KUKA KRL program: sKontur5.src, sKontur5.dat

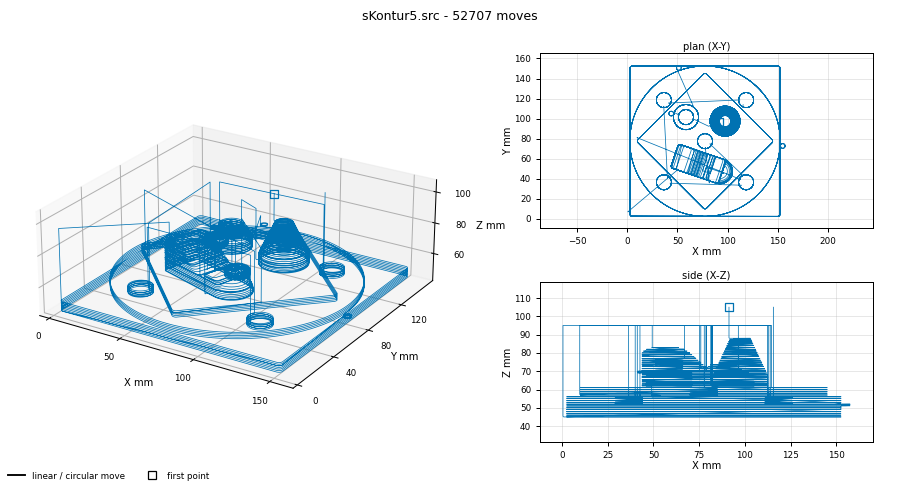
[picture p0: tool path of sKontur5.src, 52707 of 52708 moves have a stored position in this frame; points joined in program order, loops and branches not executed]
--- sKontur5.src ---
&ACCESS RVO
DEF sKontur5()
; Generated by AUTODESK Fusion 360 CAM 2.0.14793
; Creation date: Thursday, March 16, 2023 18:51:27
;FOLD sKontur5
; Start position (joint) = {A1 5,A2 -80,A3 100,A4 75,A5 -60,A6 -65}
; Tool Number            = 4
; Base Number            = 1
; Spindle Speed          = 5000 RPM
; Program file name      = sKontur5.src

PTP {A1 5,A2 -80,A3 100,A4 75,A5 -60,A6 -65,E1 0,E2 0,E3 0,E4 0,E5 0,E6 0}
LIN {X 91.288,Y 96.306,Z 105.000,A 180.000,B 0.000,C 180.000} C_DIS
LIN {X 91.288,Y 96.306,Z 90.497,A 180.000,B 0.000,C 180.000} C_DIS
; Plunge Move Starts
$VEL.CP=0.01
LIN {X 91.288,Y 96.306,Z 89.476,A 180.000,B 0.000,C 180.000} C_DIS
; Lead In Move Starts
LIN {X 91.288,Y 96.306,Z 88.351,A 180.000,B 0.000,C 180.000} C_DIS
LIN {X 91.390,Y 96.319,Z 88.103,A 180.000,B 0.000,C 180.000} C_DIS
LIN {X 91.636,Y 96.350,Z 88.000,A 180.000,B 0.000,C 180.000} C_DIS
LIN {X 91.969,Y 96.540,Z 88.000,A 180.000,B 0.000,C 180.000} C_DIS
LIN {X 92.070,Y 96.909,Z 88.000,A 180.000,B 0.000,C 180.000} C_DIS
; Cutting Move Starts
$VEL.CP=0.02
LIN {X 92.051,Y 97.075,Z 88.000,A 180.000,B 0.000,C 180.000} C_DIS
LIN {X 92.040,Y 97.254,Z 88.000,A 180.000,B 0.000,C 180.000} C_DIS
LIN {X 92.038,Y 97.433,Z 88.000,A 180.000,B 0.000,C 180.000} C_DIS
LIN {X 92.038,Y 97.612,Z 88.000,A 180.000,B 0.000,C 180.000} C_DIS
LIN {X 92.042,Y 97.790,Z 88.000,A 180.000,B 0.000,C 180.000} C_DIS
LIN {X 92.055,Y 97.969,Z 88.000,A 180.000,B 0.000,C 180.000} C_DIS
LIN {X 92.070,Y 98.091,Z 88.000,A 180.000,B 0.000,C 180.000} C_DIS
LIN {X 92.099,Y 98.327,Z 88.000,A 180.000,B 0.000,C 180.000} C_DIS
LIN {X 92.127,Y 98.505,Z 88.000,A 180.000,B 0.000,C 180.000} C_DIS
LIN {X 92.166,Y 98.684,Z 88.000,A 180.000,B 0.000,C 180.000} C_DIS
LIN {X 92.211,Y 98.863,Z 88.000,A 180.000,B 0.000,C 180.000} C_DIS
LIN {X 92.249,Y 99.007,Z 88.000,A 180.000,B 0.000,C 180.000} C_DIS
LIN {X 92.257,Y 99.042,Z 88.000,A 180.000,B 0.000,C 180.000} C_DIS
LIN {X 92.312,Y 99.221,Z 88.000,A 180.000,B 0.000,C 180.000} C_DIS
LIN {X 92.378,Y 99.399,Z 88.000,A 180.000,B 0.000,C 180.000} C_DIS
LIN {X 92.449,Y 99.578,Z 88.000,A 180.000,B 0.000,C 180.000} C_DIS
LIN {X 92.522,Y 99.757,Z 88.000,A 180.000,B 0.000,C 180.000} C_DIS
LIN {X 92.606,Y 99.932,Z 88.000,A 180.000,B 0.000,C 180.000} C_DIS
LIN {X 92.608,Y 99.936,Z 88.000,A 180.000,B 0.000,C 180.000} C_DIS
LIN {X 92.705,Y 100.114,Z 88.000,A 180.000,B 0.000,C 180.000} C_DIS
LIN {X 92.785,Y 100.260,Z 88.000,A 180.000,B 0.000,C 180.000} C_DIS
LIN {X 92.803,Y 100.293,Z 88.000,A 180.000,B 0.000,C 180.000} C_DIS
LIN {X 92.913,Y 100.472,Z 88.000,A 180.000,B 0.000,C 180.000} C_DIS
LIN {X 92.964,Y 100.547,Z 88.000,A 180.000,B 0.000,C 180.000} C_DIS
LIN {X 93.038,Y 100.651,Z 88.000,A 180.000,B 0.000,C 180.000} C_DIS
LIN {X 93.168,Y 100.829,Z 88.000,A 180.000,B 0.000,C 180.000} C_DIS
LIN {X 93.308,Y 101.008,Z 88.000,A 180.000,B 0.000,C 180.000} C_DIS
LIN {X 93.321,Y 101.023,Z 88.000,A 180.000,B 0.000,C 180.000} C_DIS
LIN {X 93.470,Y 101.187,Z 88.000,A 180.000,B 0.000,C 180.000} C_DIS
LIN {X 93.500,Y 101.218,Z 88.000,A 180.000,B 0.000,C 180.000} C_DIS
LIN {X 93.638,Y 101.366,Z 88.000,A 180.000,B 0.000,C 180.000} C_DIS
LIN {X 93.679,Y 101.407,Z 88.000,A 180.000,B 0.000,C 180.000} C_DIS
LIN {X 93.824,Y 101.545,Z 88.000,A 180.000,B 0.000,C 180.000} C_DIS
LIN {X 93.857,Y 101.574,Z 88.000,A 180.000,B 0.000,C 180.000} C_DIS
LIN {X 94.037,Y 101.723,Z 88.000,A 180.000,B 0.000,C 180.000} C_DIS
LIN {X 94.215,Y 101.868,Z 88.000,A 180.000,B 0.000,C 180.000} C_DIS
LIN {X 94.260,Y 101.902,Z 88.000,A 180.000,B 0.000,C 180.000} C_DIS
LIN {X 94.394,Y 101.996,Z 88.000,A 180.000,B 0.000,C 180.000} C_DIS
LIN {X 94.525,Y 102.081,Z 88.000,A 180.000,B 0.000,C 180.000} C_DIS
LIN {X 94.573,Y 102.111,Z 88.000,A 180.000,B 0.000,C 180.000} C_DIS
LIN {X 94.751,Y 102.223,Z 88.000,A 180.000,B 0.000,C 180.000} C_DIS
LIN {X 94.813,Y 102.260,Z 88.000,A 180.000,B 0.000,C 180.000} C_DIS
LIN {X 94.930,Y 102.324,Z 88.000,A 180.000,B 0.000,C 180.000} C_DIS
LIN {X 95.109,Y 102.411,Z 88.000,A 180.000,B 0.000,C 180.000} C_DIS
LIN {X 95.288,Y 102.495,Z 88.000,A 180.000,B 0.000,C 180.000} C_DIS
LIN {X 95.466,Y 102.574,Z 88.000,A 180.000,B 0.000,C 180.000} C_DIS
LIN {X 95.580,Y 102.617,Z 88.000,A 180.000,B 0.000,C 180.000} C_DIS
LIN {X 95.645,Y 102.640,Z 88.000,A 180.000,B 0.000,C 180.000} C_DIS
LIN {X 95.824,Y 102.698,Z 88.000,A 180.000,B 0.000,C 180.000} C_DIS
LIN {X 96.003,Y 102.756,Z 88.000,A 180.000,B 0.000,C 180.000} C_DIS
LIN {X 96.147,Y 102.796,Z 88.000,A 180.000,B 0.000,C 180.000} C_DIS
LIN {X 96.181,Y 102.805,Z 88.000,A 180.000,B 0.000,C 180.000} C_DIS
LIN {X 96.360,Y 102.843,Z 88.000,A 180.000,B 0.000,C 180.000} C_DIS
LIN {X 96.539,Y 102.877,Z 88.000,A 180.000,B 0.000,C 180.000} C_DIS
LIN {X 96.718,Y 102.909,Z 88.000,A 180.000,B 0.000,C 180.000} C_DIS
LIN {X 96.897,Y 102.932,Z 88.000,A 180.000,B 0.000,C 180.000} C_DIS
LIN {X 97.075,Y 102.946,Z 88.000,A 180.000,B 0.000,C 180.000} C_DIS
LIN {X 97.254,Y 102.957,Z 88.000,A 180.000,B 0.000,C 180.000} C_DIS
LIN {X 97.433,Y 102.965,Z 88.000,A 180.000,B 0.000,C 180.000} C_DIS
LIN {X 97.612,Y 102.964,Z 88.000,A 180.000,B 0.000,C 180.000} C_DIS
LIN {X 97.790,Y 102.954,Z 88.000,A 180.000,B 0.000,C 180.000} C_DIS
LIN {X 97.969,Y 102.943,Z 88.000,A 180.000,B 0.000,C 180.000} C_DIS
LIN {X 98.148,Y 102.928,Z 88.000,A 180.000,B 0.000,C 180.000} C_DIS
LIN {X 98.327,Y 102.902,Z 88.000,A 180.000,B 0.000,C 180.000} C_DIS
LIN {X 98.505,Y 102.868,Z 88.000,A 180.000,B 0.000,C 180.000} C_DIS
LIN {X 98.684,Y 102.834,Z 88.000,A 180.000,B 0.000,C 180.000} C_DIS
LIN {X 98.853,Y 102.796,Z 88.000,A 180.000,B 0.000,C 180.000} C_DIS
LIN {X 98.863,Y 102.793,Z 88.000,A 180.000,B 0.000,C 180.000} C_DIS
LIN {X 99.042,Y 102.742,Z 88.000,A 180.000,B 0.000,C 180.000} C_DIS
LIN {X 99.221,Y 102.683,Z 88.000,A 180.000,B 0.000,C 180.000} C_DIS
LIN {X 99.399,Y 102.625,Z 88.000,A 180.000,B 0.000,C 180.000} C_DIS
LIN {X 99.420,Y 102.617,Z 88.000,A 180.000,B 0.000,C 180.000} C_DIS
LIN {X 99.578,Y 102.555,Z 88.000,A 180.000,B 0.000,C 180.000} C_DIS
LIN {X 99.757,Y 102.474,Z 88.000,A 180.000,B 0.000,C 180.000} C_DIS
LIN {X 99.936,Y 102.390,Z 88.000,A 180.000,B 0.000,C 180.000} C_DIS
LIN {X 100.114,Y 102.300,Z 88.000,A 180.000,B 0.000,C 180.000} C_DIS
LIN {X 100.187,Y 102.260,Z 88.000,A 180.000,B 0.000,C 180.000} C_DIS
LIN {X 100.293,Y 102.196,Z 88.000,A 180.000,B 0.000,C 180.000} C_DIS
LIN {X 100.475,Y 102.081,Z 88.000,A 180.000,B 0.000,C 180.000} C_DIS
LIN {X 100.651,Y 101.966,Z 88.000,A 180.000,B 0.000,C 180.000} C_DIS
LIN {X 100.740,Y 101.902,Z 88.000,A 180.000,B 0.000,C 180.000} C_DIS
LIN {X 100.829,Y 101.833,Z 88.000,A 180.000,B 0.000,C 180.000} C_DIS
LIN {X 100.963,Y 101.723,Z 88.000,A 180.000,B 0.000,C 180.000} C_DIS
LIN {X 101.008,Y 101.686,Z 88.000,A 180.000,B 0.000,C 180.000} C_DIS
LIN {X 101.176,Y 101.545,Z 88.000,A 180.000,B 0.000,C 180.000} C_DIS
LIN {X 101.187,Y 101.535,Z 88.000,A 180.000,B 0.000,C 180.000} C_DIS
LIN {X 101.362,Y 101.366,Z 88.000,A 180.000,B 0.000,C 180.000} C_DIS
LIN {X 101.366,Y 101.361,Z 88.000,A 180.000,B 0.000,C 180.000} C_DIS
LIN {X 101.530,Y 101.187,Z 88.000,A 180.000,B 0.000,C 180.000} C_DIS
LIN {X 101.545,Y 101.171,Z 88.000,A 180.000,B 0.000,C 180.000} C_DIS
LIN {X 101.692,Y 101.008,Z 88.000,A 180.000,B 0.000,C 180.000} C_DIS
LIN {X 101.723,Y 100.970,Z 88.000,A 180.000,B 0.000,C 180.000} C_DIS
LIN {X 101.832,Y 100.829,Z 88.000,A 180.000,B 0.000,C 180.000} C_DIS
LIN {X 101.962,Y 100.651,Z 88.000,A 180.000,B 0.000,C 180.000} C_DIS
LIN {X 102.081,Y 100.482,Z 88.000,A 180.000,B 0.000,C 180.000} C_DIS
LIN {X 102.087,Y 100.472,Z 88.000,A 180.000,B 0.000,C 180.000} C_DIS
LIN {X 102.197,Y 100.293,Z 88.000,A 180.000,B 0.000,C 180.000} C_DIS
LIN {X 102.260,Y 100.179,Z 88.000,A 180.000,B 0.000,C 180.000} C_DIS
LIN {X 102.295,Y 100.114,Z 88.000,A 180.000,B 0.000,C 180.000} C_DIS
LIN {X 102.392,Y 99.936,Z 88.000,A 180.000,B 0.000,C 180.000} C_DIS
LIN {X 102.438,Y 99.844,Z 88.000,A 180.000,B 0.000,C 180.000} C_DIS
LIN {X 102.478,Y 99.757,Z 88.000,A 180.000,B 0.000,C 180.000} C_DIS
LIN {X 102.551,Y 99.578,Z 88.000,A 180.000,B 0.000,C 180.000} C_DIS
LIN {X 102.622,Y 99.399,Z 88.000,A 180.000,B 0.000,C 180.000} C_DIS
LIN {X 102.688,Y 99.221,Z 88.000,A 180.000,B 0.000,C 180.000} C_DIS
LIN {X 102.743,Y 99.042,Z 88.000,A 180.000,B 0.000,C 180.000} C_DIS
LIN {X 102.789,Y 98.863,Z 88.000,A 180.000,B 0.000,C 180.000} C_DIS
LIN {X 102.796,Y 98.834,Z 88.000,A 180.000,B 0.000,C 180.000} C_DIS
LIN {X 102.834,Y 98.684,Z 88.000,A 180.000,B 0.000,C 180.000} C_DIS
LIN {X 102.873,Y 98.505,Z 88.000,A 180.000,B 0.000,C 180.000} C_DIS
LIN {X 102.901,Y 98.327,Z 88.000,A 180.000,B 0.000,C 180.000} C_DIS
LIN {X 102.923,Y 98.148,Z 88.000,A 180.000,B 0.000,C 180.000} C_DIS
LIN {X 102.945,Y 97.969,Z 88.000,A 180.000,B 0.000,C 180.000} C_DIS
LIN {X 102.958,Y 97.790,Z 88.000,A 180.000,B 0.000,C 180.000} C_DIS
LIN {X 102.962,Y 97.612,Z 88.000,A 180.000,B 0.000,C 180.000} C_DIS
LIN {X 102.962,Y 97.433,Z 88.000,A 180.000,B 0.000,C 180.000} C_DIS
LIN {X 102.960,Y 97.254,Z 88.000,A 180.000,B 0.000,C 180.000} C_DIS
LIN {X 102.949,Y 97.075,Z 88.000,A 180.000,B 0.000,C 180.000} C_DIS
LIN {X 102.929,Y 96.897,Z 88.000,A 180.000,B 0.000,C 180.000} C_DIS
LIN {X 102.906,Y 96.718,Z 88.000,A 180.000,B 0.000,C 180.000} C_DIS
LIN {X 102.881,Y 96.539,Z 88.000,A 180.000,B 0.000,C 180.000} C_DIS
LIN {X 102.845,Y 96.360,Z 88.000,A 180.000,B 0.000,C 180.000} C_DIS
LIN {X 102.800,Y 96.181,Z 88.000,A 180.000,B 0.000,C 180.000} C_DIS
LIN {X 102.754,Y 96.003,Z 88.000,A 180.000,B 0.000,C 180.000} C_DIS
LIN {X 102.703,Y 95.824,Z 88.000,A 180.000,B 0.000,C 180.000} C_DIS
LIN {X 102.639,Y 95.645,Z 88.000,A 180.000,B 0.000,C 180.000} C_DIS
LIN {X 102.617,Y 95.588,Z 88.000,A 180.000,B 0.000,C 180.000} C_DIS
LIN {X 102.569,Y 95.466,Z 88.000,A 180.000,B 0.000,C 180.000} C_DIS
LIN {X 102.497,Y 95.288,Z 88.000,A 180.000,B 0.000,C 180.000} C_DIS
LIN {X 102.438,Y 95.156,Z 88.000,A 180.000,B 0.000,C 180.000} C_DIS
LIN {X 102.415,Y 95.109,Z 88.000,A 180.000,B 0.000,C 180.000} C_DIS
LIN {X 102.320,Y 94.930,Z 88.000,A 180.000,B 0.000,C 180.000} C_DIS
LIN {X 102.221,Y 94.751,Z 88.000,A 180.000,B 0.000,C 180.000} C_DIS
LIN {X 102.116,Y 94.573,Z 88.000,A 180.000,B 0.000,C 180.000} C_DIS
LIN {X 102.081,Y 94.518,Z 88.000,A 180.000,B 0.000,C 180.000} C_DIS
LIN {X 101.994,Y 94.394,Z 88.000,A 180.000,B 0.000,C 180.000} C_DIS
LIN {X 101.864,Y 94.215,Z 88.000,A 180.000,B 0.000,C 180.000} C_DIS
LIN {X 101.729,Y 94.036,Z 88.000,A 180.000,B 0.000,C 180.000} C_DIS
LIN {X 101.723,Y 94.030,Z 88.000,A 180.000,B 0.000,C 180.000} C_DIS
LIN {X 101.571,Y 93.857,Z 88.000,A 180.000,B 0.000,C 180.000} C_DIS
LIN {X 101.404,Y 93.679,Z 88.000,A 180.000,B 0.000,C 180.000} C_DIS
LIN {X 101.366,Y 93.639,Z 88.000,A 180.000,B 0.000,C 180.000} C_DIS
LIN {X 101.225,Y 93.500,Z 88.000,A 180.000,B 0.000,C 180.000} C_DIS
LIN {X 101.187,Y 93.465,Z 88.000,A 180.000,B 0.000,C 180.000} C_DIS
LIN {X 101.017,Y 93.321,Z 88.000,A 180.000,B 0.000,C 180.000} C_DIS
LIN {X 101.008,Y 93.314,Z 88.000,A 180.000,B 0.000,C 180.000} C_DIS
LIN {X 100.829,Y 93.167,Z 88.000,A 180.000,B 0.000,C 180.000} C_DIS
LIN {X 100.799,Y 93.142,Z 88.000,A 180.000,B 0.000,C 180.000} C_DIS
LIN {X 100.651,Y 93.034,Z 88.000,A 180.000,B 0.000,C 180.000} C_DIS
LIN {X 100.545,Y 92.964,Z 88.000,A 180.000,B 0.000,C 180.000} C_DIS
LIN {X 100.293,Y 92.804,Z 88.000,A 180.000,B 0.000,C 180.000} C_DIS
LIN {X 100.262,Y 92.785,Z 88.000,A 180.000,B 0.000,C 180.000} C_DIS
LIN {X 100.114,Y 92.700,Z 88.000,A 180.000,B 0.000,C 180.000} C_DIS
LIN {X 99.936,Y 92.610,Z 88.000,A 180.000,B 0.000,C 180.000} C_DIS
LIN {X 99.757,Y 92.526,Z 88.000,A 180.000,B 0.000,C 180.000} C_DIS
LIN {X 99.578,Y 92.445,Z 88.000,A 180.000,B 0.000,C 180.000} C_DIS
LIN {X 99.537,Y 92.427,Z 88.000,A 180.000,B 0.000,C 180.000} C_DIS
LIN {X 99.399,Y 92.375,Z 88.000,A 180.000,B 0.000,C 180.000} C_DIS
LIN {X 99.221,Y 92.317,Z 88.000,A 180.000,B 0.000,C 180.000} C_DIS
LIN {X 99.042,Y 92.258,Z 88.000,A 180.000,B 0.000,C 180.000} C_DIS
LIN {X 99.010,Y 92.249,Z 88.000,A 180.000,B 0.000,C 180.000} C_DIS
LIN {X 98.863,Y 92.207,Z 88.000,A 180.000,B 0.000,C 180.000} C_DIS
LIN {X 98.684,Y 92.166,Z 88.000,A 180.000,B 0.000,C 180.000} C_DIS
LIN {X 98.505,Y 92.132,Z 88.000,A 180.000,B 0.000,C 180.000} C_DIS
LIN {X 98.327,Y 92.098,Z 88.000,A 180.000,B 0.000,C 180.000} C_DIS
LIN {X 98.148,Y 92.072,Z 88.000,A 180.000,B 0.000,C 180.000} C_DIS
LIN {X 98.124,Y 92.070,Z 88.000,A 180.000,B 0.000,C 180.000} C_DIS
LIN {X 97.969,Y 92.057,Z 88.000,A 180.000,B 0.000,C 180.000} C_DIS
LIN {X 97.790,Y 92.046,Z 88.000,A 180.000,B 0.000,C 180.000} C_DIS
LIN {X 97.612,Y 92.036,Z 88.000,A 180.000,B 0.000,C 180.000} C_DIS
LIN {X 97.433,Y 92.035,Z 88.000,A 180.000,B 0.000,C 180.000} C_DIS
LIN {X 97.254,Y 92.043,Z 88.000,A 180.000,B 0.000,C 180.000} C_DIS
LIN {X 97.075,Y 92.054,Z 88.000,A 180.000,B 0.000,C 180.000} C_DIS
LIN {X 96.897,Y 92.068,Z 88.000,A 180.000,B 0.000,C 180.000} C_DIS
LIN {X 96.876,Y 92.070,Z 88.000,A 180.000,B 0.000,C 180.000} C_DIS
LIN {X 96.718,Y 92.091,Z 88.000,A 180.000,B 0.000,C 180.000} C_DIS
LIN {X 96.539,Y 92.123,Z 88.000,A 180.000,B 0.000,C 180.000} C_DIS
LIN {X 96.360,Y 92.157,Z 88.000,A 180.000,B 0.000,C 180.000} C_DIS
LIN {X 96.181,Y 92.195,Z 88.000,A 180.000,B 0.000,C 180.000} C_DIS
LIN {X 96.003,Y 92.244,Z 88.000,A 180.000,B 0.000,C 180.000} C_DIS
LIN {X 95.990,Y 92.249,Z 88.000,A 180.000,B 0.000,C 180.000} C_DIS
LIN {X 95.824,Y 92.302,Z 88.000,A 180.000,B 0.000,C 180.000} C_DIS
LIN {X 95.645,Y 92.360,Z 88.000,A 180.000,B 0.000,C 180.000} C_DIS
LIN {X 95.466,Y 92.426,Z 88.000,A 180.000,B 0.000,C 180.000} C_DIS
LIN {X 95.463,Y 92.427,Z 88.000,A 180.000,B 0.000,C 180.000} C_DIS
LIN {X 95.288,Y 92.505,Z 88.000,A 180.000,B 0.000,C 180.000} C_DIS
LIN {X 95.073,Y 92.606,Z 88.000,A 180.000,B 0.000,C 180.000} C_DIS
LIN {X 94.930,Y 92.676,Z 88.000,A 180.000,B 0.000,C 180.000} C_DIS
LIN {X 94.751,Y 92.777,Z 88.000,A 180.000,B 0.000,C 180.000} C_DIS
LIN {X 94.738,Y 92.785,Z 88.000,A 180.000,B 0.000,C 180.000} C_DIS
LIN {X 94.573,Y 92.889,Z 88.000,A 180.000,B 0.000,C 180.000} C_DIS
LIN {X 94.455,Y 92.964,Z 88.000,A 180.000,B 0.000,C 180.000} C_DIS
LIN {X 94.394,Y 93.004,Z 88.000,A 180.000,B 0.000,C 180.000} C_DIS
LIN {X 94.215,Y 93.132,Z 88.000,A 180.000,B 0.000,C 180.000} C_DIS
LIN {X 94.201,Y 93.142,Z 88.000,A 180.000,B 0.000,C 180.000} C_DIS
LIN {X 94.036,Y 93.277,Z 88.000,A 180.000,B 0.000,C 180.000} C_DIS
LIN {X 93.983,Y 93.321,Z 88.000,A 180.000,B 0.000,C 180.000} C_DIS
LIN {X 93.857,Y 93.426,Z 88.000,A 180.000,B 0.000,C 180.000} C_DIS
LIN {X 93.775,Y 93.500,Z 88.000,A 180.000,B 0.000,C 180.000} C_DIS
LIN {X 93.679,Y 93.593,Z 88.000,A 180.000,B 0.000,C 180.000} C_DIS
LIN {X 93.596,Y 93.679,Z 88.000,A 180.000,B 0.000,C 180.000} C_DIS
LIN {X 93.429,Y 93.857,Z 88.000,A 180.000,B 0.000,C 180.000} C_DIS
LIN {X 93.321,Y 93.977,Z 88.000,A 180.000,B 0.000,C 180.000} C_DIS
LIN {X 93.271,Y 94.036,Z 88.000,A 180.000,B 0.000,C 180.000} C_DIS
LIN {X 93.142,Y 94.206,Z 88.000,A 180.000,B 0.000,C 180.000} C_DIS
LIN {X 93.006,Y 94.394,Z 88.000,A 180.000,B 0.000,C 180.000} C_DIS
LIN {X 92.964,Y 94.453,Z 88.000,A 180.000,B 0.000,C 180.000} C_DIS
LIN {X 92.884,Y 94.573,Z 88.000,A 180.000,B 0.000,C 180.000} C_DIS
LIN {X 92.785,Y 94.740,Z 88.000,A 180.000,B 0.000,C 180.000} C_DIS
LIN {X 92.680,Y 94.930,Z 88.000,A 180.000,B 0.000,C 180.000} C_DIS
LIN {X 92.606,Y 95.068,Z 88.000,A 180.000,B 0.000,C 180.000} C_DIS
LIN {X 92.585,Y 95.109,Z 88.000,A 180.000,B 0.000,C 180.000} C_DIS
LIN {X 92.503,Y 95.288,Z 88.000,A 180.000,B 0.000,C 180.000} C_DIS
LIN {X 92.431,Y 95.466,Z 88.000,A 180.000,B 0.000,C 180.000} C_DIS
LIN {X 92.427,Y 95.476,Z 88.000,A 180.000,B 0.000,C 180.000} C_DIS
LIN {X 92.361,Y 95.645,Z 88.000,A 180.000,B 0.000,C 180.000} C_DIS
LIN {X 92.297,Y 95.824,Z 88.000,A 180.000,B 0.000,C 180.000} C_DIS
LIN {X 92.249,Y 95.993,Z 88.000,A 180.000,B 0.000,C 180.000} C_DIS
LIN {X 92.246,Y 96.003,Z 88.000,A 180.000,B 0.000,C 180.000} C_DIS
LIN {X 92.200,Y 96.181,Z 88.000,A 180.000,B 0.000,C 180.000} C_DIS
LIN {X 92.155,Y 96.360,Z 88.000,A 180.000,B 0.000,C 180.000} C_DIS
LIN {X 92.119,Y 96.539,Z 88.000,A 180.000,B 0.000,C 180.000} C_DIS
LIN {X 92.094,Y 96.718,Z 88.000,A 180.000,B 0.000,C 180.000} C_DIS
LIN {X 92.070,Y 96.909,Z 88.000,A 180.000,B 0.000,C 180.000} C_DIS
; Link Move Starts
LIN {X 92.043,Y 97.188,Z 88.000,A 180.000,B 0.000,C 180.000} C_DIS
LIN {X 92.038,Y 97.479,Z 87.999,A 180.000,B 0.000,C 180.000} C_DIS
LIN {X 92.040,Y 97.771,Z 87.998,A 180.000,B 0.000,C 180.000} C_DIS
LIN {X 92.064,Y 98.056,Z 87.997,A 180.000,B 0.000,C 180.000} C_DIS
LIN {X 92.101,Y 98.357,Z 87.995,A 180.000,B 0.000,C 180.000} C_DIS
LIN {X 92.148,Y 98.627,Z 87.993,A 180.000,B 0.000,C 180.000} C_DIS
LIN {X 92.221,Y 98.920,Z 87.990,A 180.000,B 0.000,C 180.000} C_DIS
LIN {X 92.298,Y 99.199,Z 87.987,A 180.000,B 0.000,C 180.000} C_DIS
LIN {X 92.396,Y 99.465,Z 87.984,A 180.000,B 0.000,C 180.000} C_DIS
LIN {X 92.506,Y 99.743,Z 87.980,A 180.000,B 0.000,C 180.000} C_DIS
LIN {X 92.627,Y 99.996,Z 87.976,A 180.000,B 0.000,C 180.000} C_DIS
LIN {X 92.770,Y 100.260,Z 87.972,A 180.000,B 0.000,C 180.000} C_DIS
LIN {X 92.916,Y 100.505,Z 87.967,A 180.000,B 0.000,C 180.000} C_DIS
LIN {X 93.000,Y 100.626,Z 87.964,A 180.000,B 0.000,C 180.000} C_DIS
LIN {X 93.086,Y 100.747,Z 87.962,A 180.000,B 0.000,C 180.000} C_DIS
LIN {X 93.171,Y 100.865,Z 87.959,A 180.000,B 0.000,C 180.000} C_DIS
LIN {X 93.259,Y 100.980,Z 87.956,A 180.000,B 0.000,C 180.000} C_DIS
LIN {X 93.351,Y 101.090,Z 87.954,A 180.000,B 0.000,C 180.000} C_DIS
LIN {X 93.448,Y 101.196,Z 87.951,A 180.000,B 0.000,C 180.000} C_DIS
LIN {X 93.547,Y 101.304,Z 87.948,A 180.000,B 0.000,C 180.000} C_DIS
LIN {X 93.646,Y 101.411,Z 87.945,A 180.000,B 0.000,C 180.000} C_DIS
LIN {X 93.746,Y 101.511,Z 87.941,A 180.000,B 0.000,C 180.000} C_DIS
LIN {X 93.851,Y 101.606,Z 87.938,A 180.000,B 0.000,C 180.000} C_DIS
LIN {X 93.969,Y 101.707,Z 87.935,A 180.000,B 0.000,C 180.000} C_DIS
LIN {X 94.088,Y 101.807,Z 87.931,A 180.000,B 0.000,C 180.000} C_DIS
LIN {X 94.193,Y 101.894,Z 87.928,A 180.000,B 0.000,C 180.000} C_DIS
LIN {X 94.301,Y 101.976,Z 87.925,A 180.000,B 0.000,C 180.000} C_DIS
LIN {X 94.427,Y 102.062,Z 87.921,A 180.000,B 0.000,C 180.000} C_DIS
LIN {X 94.554,Y 102.145,Z 87.917,A 180.000,B 0.000,C 180.000} C_DIS
LIN {X 94.674,Y 102.223,Z 87.913,A 180.000,B 0.000,C 180.000} C_DIS
LIN {X 94.795,Y 102.298,Z 87.910,A 180.000,B 0.000,C 180.000} C_DIS
LIN {X 94.922,Y 102.369,Z 87.906,A 180.000,B 0.000,C 180.000} C_DIS
LIN {X 95.052,Y 102.435,Z 87.902,A 180.000,B 0.000,C 180.000} C_DIS
LIN {X 95.190,Y 102.502,Z 87.898,A 180.000,B 0.000,C 180.000} C_DIS
LIN {X 95.329,Y 102.569,Z 87.893,A 180.000,B 0.000,C 180.000} C_DIS
LIN {X 95.461,Y 102.627,Z 87.889,A 180.000,B 0.000,C 180.000} C_DIS
LIN {X 95.596,Y 102.680,Z 87.885,A 180.000,B 0.000,C 180.000} C_DIS
LIN {X 95.736,Y 102.728,Z 87.881,A 180.000,B 0.000,C 180.000} C_DIS
LIN {X 95.875,Y 102.775,Z 87.876,A 180.000,B 0.000,C 180.000} C_DIS
LIN {X 96.010,Y 102.820,Z 87.872,A 180.000,B 0.000,C 180.000} C_DIS
LIN {X 96.146,Y 102.859,Z 87.868,A 180.000,B 0.000,C 180.000} C_DIS
LIN {X 96.290,Y 102.894,Z 87.863,A 180.000,B 0.000,C 180.000} C_DIS
LIN {X 96.436,Y 102.924,Z 87.859,A 180.000,B 0.000,C 180.000} C_DIS
LIN {X 96.584,Y 102.955,Z 87.854,A 180.000,B 0.000,C 180.000} C_DIS
LIN {X 96.733,Y 102.983,Z 87.849,A 180.000,B 0.000,C 180.000} C_DIS
LIN {X 96.872,Y 103.003,Z 87.844,A 180.000,B 0.000,C 180.000} C_DIS
LIN {X 97.011,Y 103.017,Z 87.840,A 180.000,B 0.000,C 180.000} C_DIS
LIN {X 97.087,Y 103.022,Z 87.837,A 180.000,B 0.000,C 180.000} C_DIS
LIN {X 97.163,Y 103.028,Z 87.835,A 180.000,B 0.000,C 180.000} C_DIS
LIN {X 97.238,Y 103.034,Z 87.832,A 180.000,B 0.000,C 180.000} C_DIS
LIN {X 97.314,Y 103.040,Z 87.830,A 180.000,B 0.000,C 180.000} C_DIS
LIN {X 97.457,Y 103.048,Z 87.825,A 180.000,B 0.000,C 180.000} C_DIS
LIN {X 97.601,Y 103.048,Z 87.820,A 180.000,B 0.000,C 180.000} C_DIS
LIN {X 97.677,Y 103.047,Z 87.817,A 180.000,B 0.000,C 180.000} C_DIS
LIN {X 97.752,Y 103.043,Z 87.815,A 180.000,B 0.000,C 180.000} C_DIS
LIN {X 97.976,Y 103.033,Z 87.807,A 180.000,B 0.000,C 180.000} C_DIS
LIN {X 98.049,Y 103.029,Z 87.804,A 180.000,B 0.000,C 180.000} C_DIS
LIN {X 98.122,Y 103.023,Z 87.802,A 180.000,B 0.000,C 180.000} C_DIS
LIN {X 98.195,Y 103.016,Z 87.799,A 180.000,B 0.000,C 180.000} C_DIS
LIN {X 98.267,Y 103.007,Z 87.797,A 180.000,B 0.000,C 180.000} C_DIS
LIN {X 98.339,Y 102.997,Z 87.794,A 180.000,B 0.000,C 180.000} C_DIS
LIN {X 98.411,Y 102.985,Z 87.792,A 180.000,B 0.000,C 180.000} C_DIS
LIN {X 98.483,Y 102.973,Z 87.789,A 180.000,B 0.000,C 180.000} C_DIS
LIN {X 98.633,Y 102.947,Z 87.784,A 180.000,B 0.000,C 180.000} C_DIS
LIN {X 98.708,Y 102.933,Z 87.781,A 180.000,B 0.000,C 180.000} C_DIS
LIN {X 98.783,Y 102.919,Z 87.778,A 180.000,B 0.000,C 180.000} C_DIS
LIN {X 98.922,Y 102.887,Z 87.773,A 180.000,B 0.000,C 180.000} C_DIS
LIN {X 98.992,Y 102.869,Z 87.771,A 180.000,B 0.000,C 180.000} C_DIS
LIN {X 99.060,Y 102.849,Z 87.768,A 180.000,B 0.000,C 180.000} C_DIS
LIN {X 99.133,Y 102.827,Z 87.766,A 180.000,B 0.000,C 180.000} C_DIS
LIN {X 99.279,Y 102.782,Z 87.760,A 180.000,B 0.000,C 180.000} C_DIS
LIN {X 99.352,Y 102.759,Z 87.758,A 180.000,B 0.000,C 180.000} C_DIS
LIN {X 99.421,Y 102.738,Z 87.755,A 180.000,B 0.000,C 180.000} C_DIS
LIN {X 99.490,Y 102.714,Z 87.753,A 180.000,B 0.000,C 180.000} C_DIS
LIN {X 99.558,Y 102.690,Z 87.750,A 180.000,B 0.000,C 180.000} C_DIS
LIN {X 99.625,Y 102.663,Z 87.748,A 180.000,B 0.000,C 180.000} C_DIS
LIN {X 99.694,Y 102.634,Z 87.745,A 180.000,B 0.000,C 180.000} C_DIS
LIN {X 99.763,Y 102.604,Z 87.742,A 180.000,B 0.000,C 180.000} C_DIS
LIN {X 99.966,Y 102.512,Z 87.735,A 180.000,B 0.000,C 180.000} C_DIS
LIN {X 100.032,Y 102.483,Z 87.732,A 180.000,B 0.000,C 180.000} C_DIS
LIN {X 100.098,Y 102.451,Z 87.729,A 180.000,B 0.000,C 180.000} C_DIS
LIN {X 100.163,Y 102.419,Z 87.727,A 180.000,B 0.000,C 180.000} C_DIS
LIN {X 100.229,Y 102.384,Z 87.724,A 180.000,B 0.000,C 180.000} C_DIS
LIN {X 100.294,Y 102.347,Z 87.722,A 180.000,B 0.000,C 180.000} C_DIS
LIN {X 100.358,Y 102.310,Z 87.719,A 180.000,B 0.000,C 180.000} C_DIS
LIN {X 100.422,Y 102.271,Z 87.717,A 180.000,B 0.000,C 180.000} C_DIS
LIN {X 100.550,Y 102.193,Z 87.711,A 180.000,B 0.000,C 180.000} C_DIS
LIN {X 100.614,Y 102.153,Z 87.709,A 180.000,B 0.000,C 180.000} C_DIS
LIN {X 100.677,Y 102.114,Z 87.706,A 180.000,B 0.000,C 180.000} C_DIS
LIN {X 100.739,Y 102.073,Z 87.703,A 180.000,B 0.000,C 180.000} C_DIS
LIN {X 100.800,Y 102.032,Z 87.701,A 180.000,B 0.000,C 180.000} C_DIS
LIN {X 100.859,Y 101.989,Z 87.698,A 180.000,B 0.000,C 180.000} C_DIS
LIN {X 100.918,Y 101.944,Z 87.696,A 180.000,B 0.000,C 180.000} C_DIS
LIN {X 100.978,Y 101.896,Z 87.693,A 180.000,B 0.000,C 180.000} C_DIS
LIN {X 101.099,Y 101.800,Z 87.688,A 180.000,B 0.000,C 180.000} C_DIS
LIN {X 101.159,Y 101.752,Z 87.685,A 180.000,B 0.000,C 180.000} C_DIS
LIN {X 101.215,Y 101.706,Z 87.682,A 180.000,B 0.000,C 180.000} C_DIS
LIN {X 101.271,Y 101.660,Z 87.680,A 180.000,B 0.000,C 180.000} C_DIS
LIN {X 101.326,Y 101.612,Z 87.677,A 180.000,B 0.000,C 180.000} C_DIS
LIN {X 101.379,Y 101.563,Z 87.675,A 180.000,B 0.000,C 180.000} C_DIS
LIN {X 101.434,Y 101.511,Z 87.672,A 180.000,B 0.000,C 180.000} C_DIS
LIN {X 101.486,Y 101.458,Z 87.670,A 180.000,B 0.000,C 180.000} C_DIS
LIN {X 101.539,Y 101.404,Z 87.667,A 180.000,B 0.000,C 180.000} C_DIS
LIN {X 101.643,Y 101.297,Z 87.662,A 180.000,B 0.000,C 180.000} C_DIS
LIN {X 101.695,Y 101.243,Z 87.659,A 180.000,B 0.000,C 180.000} C_DIS
LIN {X 101.747,Y 101.189,Z 87.657,A 180.000,B 0.000,C 180.000} C_DIS
LIN {X 101.797,Y 101.133,Z 87.654,A 180.000,B 0.000,C 180.000} C_DIS
LIN {X 101.846,Y 101.078,Z 87.651,A 180.000,B 0.000,C 180.000} C_DIS
LIN {X 101.893,Y 101.021,Z 87.649,A 180.000,B 0.000,C 180.000} C_DIS
LIN {X 101.938,Y 100.963,Z 87.646,A 180.000,B 0.000,C 180.000} C_DIS
LIN {X 101.983,Y 100.904,Z 87.644,A 180.000,B 0.000,C 180.000} C_DIS
LIN {X 102.122,Y 100.720,Z 87.636,A 180.000,B 0.000,C 180.000} C_DIS
LIN {X 102.167,Y 100.659,Z 87.633,A 180.000,B 0.000,C 180.000} C_DIS
LIN {X 102.210,Y 100.599,Z 87.630,A 180.000,B 0.000,C 180.000} C_DIS
LIN {X 102.251,Y 100.539,Z 87.628,A 180.000,B 0.000,C 180.000} C_DIS
LIN {X 102.291,Y 100.478,Z 87.625,A 180.000,B 0.000,C 180.000} C_DIS
LIN {X 102.329,Y 100.415,Z 87.623,A 180.000,B 0.000,C 180.000} C_DIS
LIN {X 102.368,Y 100.350,Z 87.620,A 180.000,B 0.000,C 180.000} C_DIS
LIN {X 102.518,Y 100.087,Z 87.609,A 180.000,B 0.000,C 180.000} C_DIS
LIN {X 102.554,Y 100.021,Z 87.607,A 180.000,B 0.000,C 180.000} C_DIS
LIN {X 102.589,Y 99.955,Z 87.604,A 180.000,B 0.000,C 180.000} C_DIS
LIN {X 102.623,Y 99.888,Z 87.602,A 180.000,B 0.000,C 180.000} C_DIS
LIN {X 102.654,Y 99.821,Z 87.599,A 180.000,B 0.000,C 180.000} C_DIS
LIN {X 102.684,Y 99.753,Z 87.596,A 180.000,B 0.000,C 180.000} C_DIS
LIN {X 102.713,Y 99.684,Z 87.594,A 180.000,B 0.000,C 180.000} C_DIS
LIN {X 102.801,Y 99.472,Z 87.586,A 180.000,B 0.000,C 180.000} C_DIS
LIN {X 102.830,Y 99.400,Z 87.583,A 180.000,B 0.000,C 180.000} C_DIS
LIN {X 102.858,Y 99.328,Z 87.580,A 180.000,B 0.000,C 180.000} C_DIS
LIN {X 102.882,Y 99.260,Z 87.578,A 180.000,B 0.000,C 180.000} C_DIS
LIN {X 102.905,Y 99.192,Z 87.575,A 180.000,B 0.000,C 180.000} C_DIS
LIN {X 102.927,Y 99.123,Z 87.573,A 180.000,B 0.000,C 180.000} C_DIS
LIN {X 102.946,Y 99.054,Z 87.570,A 180.000,B 0.000,C 180.000} C_DIS
LIN {X 102.967,Y 98.979,Z 87.568,A 180.000,B 0.000,C 180.000} C_DIS
LIN {X 103.028,Y 98.756,Z 87.560,A 180.000,B 0.000,C 180.000} C_DIS
LIN {X 103.047,Y 98.685,Z 87.557,A 180.000,B 0.000,C 180.000} C_DIS
LIN {X 103.064,Y 98.613,Z 87.554,A 180.000,B 0.000,C 180.000} C_DIS
LIN {X 103.079,Y 98.540,Z 87.552,A 180.000,B 0.000,C 180.000} C_DIS
LIN {X 103.093,Y 98.468,Z 87.549,A 180.000,B 0.000,C 180.000} C_DIS
LIN {X 103.105,Y 98.392,Z 87.547,A 180.000,B 0.000,C 180.000} C_DIS
LIN {X 103.116,Y 98.316,Z 87.544,A 180.000,B 0.000,C 180.000} C_DIS
LIN {X 103.149,Y 98.090,Z 87.536,A 180.000,B 0.000,C 180.000} C_DIS
LIN {X 103.159,Y 98.016,Z 87.533,A 180.000,B 0.000,C 180.000} C_DIS
LIN {X 103.167,Y 97.941,Z 87.531,A 180.000,B 0.000,C 180.000} C_DIS
LIN {X 103.174,Y 97.867,Z 87.528,A 180.000,B 0.000,C 180.000} C_DIS
LIN {X 103.180,Y 97.792,Z 87.525,A 180.000,B 0.000,C 180.000} C_DIS
LIN {X 103.183,Y 97.717,Z 87.523,A 180.000,B 0.000,C 180.000} C_DIS
LIN {X 103.185,Y 97.643,Z 87.520,A 180.000,B 0.000,C 180.000} C_DIS
LIN {X 103.189,Y 97.415,Z 87.512,A 180.000,B 0.000,C 180.000} C_DIS
LIN {X 103.190,Y 97.338,Z 87.510,A 180.000,B 0.000,C 180.000} C_DIS
LIN {X 103.190,Y 97.261,Z 87.507,A 180.000,B 0.000,C 180.000} C_DIS
LIN {X 103.189,Y 97.186,Z 87.504,A 180.000,B 0.000,C 180.000} C_DIS
LIN {X 103.185,Y 97.111,Z 87.502,A 180.000,B 0.000,C 180.000} C_DIS
LIN {X 103.180,Y 97.037,Z 87.499,A 180.000,B 0.000,C 180.000} C_DIS
LIN {X 103.174,Y 96.962,Z 87.496,A 180.000,B 0.000,C 180.000} C_DIS
LIN {X 103.165,Y 96.886,Z 87.494,A 180.000,B 0.000,C 180.000} C_DIS
LIN {X 103.140,Y 96.656,Z 87.486,A 180.000,B 0.000,C 180.000} C_DIS
LIN {X 103.131,Y 96.583,Z 87.483,A 180.000,B 0.000,C 180.000} C_DIS
LIN {X 103.122,Y 96.510,Z 87.481,A 180.000,B 0.000,C 180.000} C_DIS
LIN {X 103.110,Y 96.437,Z 87.478,A 180.000,B 0.000,C 180.000} C_DIS
LIN {X 103.096,Y 96.364,Z 87.475,A 180.000,B 0.000,C 180.000} C_DIS
LIN {X 103.081,Y 96.289,Z 87.473,A 180.000,B 0.000,C 180.000} C_DIS
LIN {X 103.063,Y 96.214,Z 87.470,A 180.000,B 0.000,C 180.000} C_DIS
LIN {X 103.010,Y 95.989,Z 87.462,A 180.000,B 0.000,C 180.000} C_DIS
LIN {X 102.992,Y 95.915,Z 87.459,A 180.000,B 0.000,C 180.000} C_DIS
LIN {X 102.973,Y 95.841,Z 87.457,A 180.000,B 0.000,C 180.000} C_DIS
LIN {X 102.952,Y 95.767,Z 87.454,A 180.000,B 0.000,C 180.000} C_DIS
LIN {X 102.930,Y 95.696,Z 87.451,A 180.000,B 0.000,C 180.000} C_DIS
LIN {X 102.907,Y 95.625,Z 87.449,A 180.000,B 0.000,C 180.000} C_DIS
LIN {X 102.882,Y 95.555,Z 87.446,A 180.000,B 0.000,C 180.000} C_DIS
LIN {X 102.856,Y 95.486,Z 87.444,A 180.000,B 0.000,C 180.000} C_DIS
LIN {X 102.773,Y 95.266,Z 87.435,A 180.000,B 0.000,C 180.000} C_DIS
LIN {X 102.745,Y 95.193,Z 87.433,A 180.000,B 0.000,C 180.000} C_DIS
LIN {X 102.716,Y 95.124,Z 87.430,A 180.000,B 0.000,C 180.000} C_DIS
LIN {X 102.686,Y 95.056,Z 87.427,A 180.000,B 0.000,C 180.000} C_DIS
LIN {X 102.655,Y 94.989,Z 87.425,A 180.000,B 0.000,C 180.000} C_DIS
LIN {X 102.622,Y 94.922,Z 87.422,A 180.000,B 0.000,C 180.000} C_DIS
LIN {X 102.587,Y 94.854,Z 87.420,A 180.000,B 0.000,C 180.000} C_DIS
LIN {X 102.478,Y 94.648,Z 87.411,A 180.000,B 0.000,C 180.000} C_DIS
LIN {X 102.443,Y 94.582,Z 87.409,A 180.000,B 0.000,C 180.000} C_DIS
LIN {X 102.406,Y 94.516,Z 87.406,A 180.000,B 0.000,C 180.000} C_DIS
LIN {X 102.368,Y 94.450,Z 87.404,A 180.000,B 0.000,C 180.000} C_DIS
LIN {X 102.328,Y 94.386,Z 87.401,A 180.000,B 0.000,C 180.000} C_DIS
LIN {X 102.287,Y 94.322,Z 87.398,A 180.000,B 0.000,C 180.000} C_DIS
LIN {X 102.244,Y 94.259,Z 87.396,A 180.000,B 0.000,C 180.000} C_DIS
LIN {X 102.201,Y 94.196,Z 87.393,A 180.000,B 0.000,C 180.000} C_DIS
LIN {X 102.113,Y 94.071,Z 87.388,A 180.000,B 0.000,C 180.000} C_DIS
LIN {X 102.068,Y 94.008,Z 87.385,A 180.000,B 0.000,C 180.000} C_DIS
LIN {X 102.023,Y 93.945,Z 87.382,A 180.000,B 0.000,C 180.000} C_DIS
LIN {X 101.977,Y 93.883,Z 87.379,A 180.000,B 0.000,C 180.000} C_DIS
LIN {X 101.930,Y 93.824,Z 87.377,A 180.000,B 0.000,C 180.000} C_DIS
LIN {X 101.882,Y 93.765,Z 87.374,A 180.000,B 0.000,C 180.000} C_DIS
LIN {X 101.833,Y 93.708,Z 87.372,A 180.000,B 0.000,C 180.000} C_DIS
LIN {X 101.782,Y 93.652,Z 87.369,A 180.000,B 0.000,C 180.000} C_DIS
LIN {X 101.628,Y 93.482,Z 87.361,A 180.000,B 0.000,C 180.000} C_DIS
LIN {X 101.577,Y 93.426,Z 87.358,A 180.000,B 0.000,C 180.000} C_DIS
LIN {X 101.525,Y 93.371,Z 87.356,A 180.000,B 0.000,C 180.000} C_DIS
LIN {X 101.471,Y 93.317,Z 87.353,A 180.000,B 0.000,C 180.000} C_DIS
LIN {X 101.416,Y 93.264,Z 87.350,A 180.000,B 0.000,C 180.000} C_DIS
LIN {X 101.360,Y 93.212,Z 87.348,A 180.000,B 0.000,C 180.000} C_DIS
LIN {X 101.302,Y 93.161,Z 87.345,A 180.000,B 0.000,C 180.000} C_DIS
LIN {X 101.243,Y 93.110,Z 87.342,A 180.000,B 0.000,C 180.000} C_DIS
LIN {X 101.067,Y 92.960,Z 87.334,A 180.000,B 0.000,C 180.000} C_DIS
LIN {X 101.009,Y 92.911,Z 87.331,A 180.000,B 0.000,C 180.000} C_DIS
LIN {X 100.950,Y 92.864,Z 87.329,A 180.000,B 0.000,C 180.000} C_DIS
LIN {X 100.890,Y 92.818,Z 87.326,A 180.000,B 0.000,C 180.000} C_DIS
LIN {X 100.828,Y 92.772,Z 87.323,A 180.000,B 0.000,C 180.000} C_DIS
LIN {X 100.764,Y 92.728,Z 87.321,A 180.000,B 0.000,C 180.000} C_DIS
LIN {X 100.700,Y 92.685,Z 87.318,A 180.000,B 0.000,C 180.000} C_DIS
LIN {X 100.635,Y 92.643,Z 87.315,A 180.000,B 0.000,C 180.000} C_DIS
LIN {X 100.507,Y 92.559,Z 87.310,A 180.000,B 0.000,C 180.000} C_DIS
LIN {X 100.443,Y 92.517,Z 87.307,A 180.000,B 0.000,C 180.000} C_DIS
LIN {X 100.378,Y 92.476,Z 87.305,A 180.000,B 0.000,C 180.000} C_DIS
LIN {X 100.312,Y 92.437,Z 87.302,A 180.000,B 0.000,C 180.000} C_DIS
LIN {X 100.245,Y 92.399,Z 87.299,A 180.000,B 0.000,C 180.000} C_DIS
LIN {X 100.177,Y 92.363,Z 87.297,A 180.000,B 0.000,C 180.000} C_DIS
LIN {X 100.109,Y 92.328,Z 87.294,A 180.000,B 0.000,C 180.000} C_DIS
LIN {X 99.969,Y 92.259,Z 87.288,A 180.000,B 0.000,C 180.000} C_DIS
LIN {X 99.899,Y 92.225,Z 87.286,A 180.000,B 0.000,C 180.000} C_DIS
LIN {X 99.829,Y 92.190,Z 87.283,A 180.000,B 0.000,C 180.000} C_DIS
LIN {X 99.759,Y 92.158,Z 87.280,A 180.000,B 0.000,C 180.000} C_DIS
LIN {X 99.689,Y 92.126,Z 87.278,A 180.000,B 0.000,C 180.000} C_DIS
LIN {X 99.618,Y 92.096,Z 87.275,A 180.000,B 0.000,C 180.000} C_DIS
LIN {X 99.547,Y 92.068,Z 87.272,A 180.000,B 0.000,C 180.000} C_DIS
LIN {X 99.475,Y 92.041,Z 87.270,A 180.000,B 0.000,C 180.000} C_DIS
LIN {X 99.402,Y 92.016,Z 87.267,A 180.000,B 0.000,C 180.000} C_DIS
LIN {X 99.184,Y 91.941,Z 87.259,A 180.000,B 0.000,C 180.000} C_DIS
LIN {X 99.111,Y 91.917,Z 87.256,A 180.000,B 0.000,C 180.000} C_DIS
LIN {X 99.038,Y 91.893,Z 87.254,A 180.000,B 0.000,C 180.000} C_DIS
LIN {X 98.965,Y 91.872,Z 87.251,A 180.000,B 0.000,C 180.000} C_DIS
LIN {X 98.890,Y 91.852,Z 87.248,A 180.000,B 0.000,C 180.000} C_DIS
LIN {X 98.815,Y 91.834,Z 87.245,A 180.000,B 0.000,C 180.000} C_DIS
LIN {X 98.740,Y 91.817,Z 87.243,A 180.000,B 0.000,C 180.000} C_DIS
LIN {X 98.664,Y 91.801,Z 87.240,A 180.000,B 0.000,C 180.000} C_DIS
LIN {X 98.511,Y 91.769,Z 87.235,A 180.000,B 0.000,C 180.000} C_DIS
LIN {X 98.434,Y 91.754,Z 87.232,A 180.000,B 0.000,C 180.000} C_DIS
LIN {X 98.357,Y 91.739,Z 87.229,A 180.000,B 0.000,C 180.000} C_DIS
LIN {X 98.282,Y 91.726,Z 87.226,A 180.000,B 0.000,C 180.000} C_DIS
LIN {X 98.207,Y 91.715,Z 87.224,A 180.000,B 0.000,C 180.000} C_DIS
LIN {X 98.131,Y 91.705,Z 87.221,A 180.000,B 0.000,C 180.000} C_DIS
LIN {X 98.055,Y 91.698,Z 87.219,A 180.000,B 0.000,C 180.000} C_DIS
LIN {X 97.977,Y 91.691,Z 87.216,A 180.000,B 0.000,C 180.000} C_DIS
LIN {X 97.822,Y 91.679,Z 87.210,A 180.000,B 0.000,C 180.000} C_DIS
LIN {X 97.744,Y 91.673,Z 87.208,A 180.000,B 0.000,C 180.000} C_DIS
LIN {X 97.667,Y 91.667,Z 87.205,A 180.000,B 0.000,C 180.000} C_DIS
LIN {X 97.590,Y 91.663,Z 87.202,A 180.000,B 0.000,C 180.000} C_DIS
LIN {X 97.512,Y 91.660,Z 87.200,A 180.000,B 0.000,C 180.000} C_DIS
LIN {X 97.435,Y 91.660,Z 87.197,A 180.000,B 0.000,C 180.000} C_DIS
LIN {X 97.357,Y 91.661,Z 87.194,A 180.000,B 0.000,C 180.000} C_DIS
LIN {X 97.280,Y 91.663,Z 87.191,A 180.000,B 0.000,C 180.000} C_DIS
LIN {X 97.125,Y 91.671,Z 87.186,A 180.000,B 0.000,C 180.000} C_DIS
LIN {X 97.047,Y 91.674,Z 87.183,A 180.000,B 0.000,C 180.000} C_DIS
LIN {X 96.969,Y 91.678,Z 87.181,A 180.000,B 0.000,C 180.000} C_DIS
LIN {X 96.892,Y 91.683,Z 87.178,A 180.000,B 0.000,C 180.000} C_DIS
LIN {X 96.814,Y 91.690,Z 87.175,A 180.000,B 0.000,C 180.000} C_DIS
LIN {X 96.738,Y 91.698,Z 87.173,A 180.000,B 0.000,C 180.000} C_DIS
LIN {X 96.661,Y 91.708,Z 87.170,A 180.000,B 0.000,C 180.000} C_DIS
LIN {X 96.585,Y 91.720,Z 87.168,A 180.000,B 0.000,C 180.000} C_DIS
LIN {X 96.508,Y 91.733,Z 87.165,A 180.000,B 0.000,C 180.000} C_DIS
LIN {X 96.431,Y 91.746,Z 87.163,A 180.000,B 0.000,C 180.000} C_DIS
LIN {X 96.354,Y 91.760,Z 87.160,A 180.000,B 0.000,C 180.000} C_DIS
LIN {X 96.277,Y 91.773,Z 87.158,A 180.000,B 0.000,C 180.000} C_DIS
LIN {X 96.200,Y 91.787,Z 87.155,A 180.000,B 0.000,C 180.000} C_DIS
LIN {X 96.048,Y 91.820,Z 87.150,A 180.000,B 0.000,C 180.000} C_DIS
LIN {X 95.898,Y 91.859,Z 87.145,A 180.000,B 0.000,C 180.000} C_DIS
LIN {X 95.749,Y 91.905,Z 87.140,A 180.000,B 0.000,C 180.000} C_DIS
LIN {X 95.599,Y 91.951,Z 87.136,A 180.000,B 0.000,C 180.000} C_DIS
LIN {X 95.452,Y 91.998,Z 87.131,A 180.000,B 0.000,C 180.000} C_DIS
LIN {X 95.306,Y 92.052,Z 87.126,A 180.000,B 0.000,C 180.000} C_DIS
LIN {X 95.162,Y 92.112,Z 87.122,A 180.000,B 0.000,C 180.000} C_DIS
LIN {X 95.019,Y 92.176,Z 87.117,A 180.000,B 0.000,C 180.000} C_DIS
LIN {X 94.877,Y 92.241,Z 87.113,A 180.000,B 0.000,C 180.000} C_DIS
LIN {X 94.737,Y 92.308,Z 87.108,A 180.000,B 0.000,C 180.000} C_DIS
LIN {X 94.599,Y 92.382,Z 87.104,A 180.000,B 0.000,C 180.000} C_DIS
LIN {X 94.464,Y 92.461,Z 87.100,A 180.000,B 0.000,C 180.000} C_DIS
LIN {X 94.330,Y 92.543,Z 87.095,A 180.000,B 0.000,C 180.000} C_DIS
LIN {X 94.197,Y 92.626,Z 87.091,A 180.000,B 0.000,C 180.000} C_DIS
LIN {X 94.067,Y 92.712,Z 87.087,A 180.000,B 0.000,C 180.000} C_DIS
LIN {X 93.940,Y 92.804,Z 87.083,A 180.000,B 0.000,C 180.000} C_DIS
LIN {X 93.818,Y 92.901,Z 87.079,A 180.000,B 0.000,C 180.000} C_DIS
LIN {X 93.696,Y 92.999,Z 87.076,A 180.000,B 0.000,C 180.000} C_DIS
LIN {X 93.575,Y 93.098,Z 87.072,A 180.000,B 0.000,C 180.000} C_DIS
LIN {X 93.458,Y 93.202,Z 87.068,A 180.000,B 0.000,C 180.000} C_DIS
LIN {X 93.345,Y 93.310,Z 87.065,A 180.000,B 0.000,C 180.000} C_DIS
LIN {X 93.236,Y 93.423,Z 87.061,A 180.000,B 0.000,C 180.000} C_DIS
LIN {X 93.127,Y 93.537,Z 87.058,A 180.000,B 0.000,C 180.000} C_DIS
LIN {X 93.019,Y 93.651,Z 87.054,A 180.000,B 0.000,C 180.000} C_DIS
LIN {X 92.918,Y 93.770,Z 87.051,A 180.000,B 0.000,C 180.000} C_DIS
LIN {X 92.821,Y 93.893,Z 87.048,A 180.000,B 0.000,C 180.000} C_DIS
LIN {X 92.727,Y 94.019,Z 87.045,A 180.000,B 0.000,C 180.000} C_DIS
LIN {X 92.634,Y 94.146,Z 87.042,A 180.000,B 0.000,C 180.000} C_DIS
LIN {X 92.544,Y 94.274,Z 87.039,A 180.000,B 0.000,C 180.000} C_DIS
LIN {X 92.459,Y 94.406,Z 87.036,A 180.000,B 0.000,C 180.000} C_DIS
LIN {X 92.379,Y 94.542,Z 87.034,A 180.000,B 0.000,C 180.000} C_DIS
LIN {X 92.303,Y 94.679,Z 87.031,A 180.000,B 0.000,C 180.000} C_DIS
LIN {X 92.154,Y 94.955,Z 87.026,A 180.000,B 0.000,C 180.000} C_DIS
LIN {X 92.028,Y 95.244,Z 87.022,A 180.000,B 0.000,C 180.000} C_DIS
LIN {X 91.912,Y 95.536,Z 87.018,A 180.000,B 0.000,C 180.000} C_DIS
LIN {X 91.860,Y 95.684,Z 87.016,A 180.000,B 0.000,C 180.000} C_DIS
LIN {X 91.814,Y 95.835,Z 87.014,A 180.000,B 0.000,C 180.000} C_DIS
LIN {X 91.734,Y 96.139,Z 87.011,A 180.000,B 0.000,C 180.000} C_DIS
LIN {X 91.666,Y 96.446,Z 87.008,A 180.000,B 0.000,C 180.000} C_DIS
LIN {X 91.621,Y 96.758,Z 87.005,A 180.000,B 0.000,C 180.000} C_DIS
LIN {X 91.585,Y 97.071,Z 87.003,A 180.000,B 0.000,C 180.000} C_DIS
LIN {X 91.573,Y 97.385,Z 87.002,A 180.000,B 0.000,C 180.000} C_DIS
LIN {X 91.573,Y 97.700,Z 87.001,A 180.000,B 0.000,C 180.000} C_DIS
LIN {X 91.591,Y 98.015,Z 87.000,A 180.000,B 0.000,C 180.000} C_DIS
LIN {X 91.616,Y 98.223,Z 87.000,A 180.000,B 0.000,C 180.000} C_DIS
; Cutting Move Starts
LIN {X 91.629,Y 98.327,Z 87.000,A 180.000,B 0.000,C 180.000} C_DIS
LIN {X 91.654,Y 98.505,Z 87.000,A 180.000,B 0.000,C 180.000} C_DIS
LIN {X 91.687,Y 98.684,Z 87.000,A 180.000,B 0.000,C 180.000} C_DIS
LIN {X 91.712,Y 98.794,Z 87.000,A 180.000,B 0.000,C 180.000} C_DIS
LIN {X 91.730,Y 98.863,Z 87.000,A 180.000,B 0.000,C 180.000} C_DIS
LIN {X 91.776,Y 99.042,Z 87.000,A 180.000,B 0.000,C 180.000} C_DIS
LIN {X 91.823,Y 99.221,Z 87.000,A 180.000,B 0.000,C 180.000} C_DIS
LIN {X 91.880,Y 99.399,Z 87.000,A 180.000,B 0.000,C 180.000} C_DIS
LIN {X 91.891,Y 99.431,Z 87.000,A 180.000,B 0.000,C 180.000} C_DIS
LIN {X 91.947,Y 99.578,Z 87.000,A 180.000,B 0.000,C 180.000} C_DIS
LIN {X 92.018,Y 99.757,Z 87.000,A 180.000,B 0.000,C 180.000} C_DIS
LIN {X 92.070,Y 99.886,Z 87.000,A 180.000,B 0.000,C 180.000} C_DIS
LIN {X 92.091,Y 99.936,Z 87.000,A 180.000,B 0.000,C 180.000} C_DIS
LIN {X 92.175,Y 100.114,Z 87.000,A 180.000,B 0.000,C 180.000} C_DIS
LIN {X 92.249,Y 100.253,Z 87.000,A 180.000,B 0.000,C 180.000} C_DIS
LIN {X 92.369,Y 100.472,Z 87.000,A 180.000,B 0.000,C 180.000} C_DIS
LIN {X 92.427,Y 100.574,Z 87.000,A 180.000,B 0.000,C 180.000} C_DIS
LIN {X 92.473,Y 100.651,Z 87.000,A 180.000,B 0.000,C 180.000} C_DIS
LIN {X 92.592,Y 100.829,Z 87.000,A 180.000,B 0.000,C 180.000} C_DIS
LIN {X 92.606,Y 100.849,Z 87.000,A 180.000,B 0.000,C 180.000} C_DIS
LIN {X 92.721,Y 101.008,Z 87.000,A 180.000,B 0.000,C 180.000} C_DIS
LIN {X 92.785,Y 101.096,Z 87.000,A 180.000,B 0.000,C 180.000} C_DIS
LIN {X 92.853,Y 101.187,Z 87.000,A 180.000,B 0.000,C 180.000} C_DIS
LIN {X 92.964,Y 101.322,Z 87.000,A 180.000,B 0.000,C 180.000} C_DIS
LIN {X 93.001,Y 101.366,Z 87.000,A 180.000,B 0.000,C 180.000} C_DIS
LIN {X 93.142,Y 101.519,Z 87.000,A 180.000,B 0.000,C 180.000} C_DIS
LIN {X 93.166,Y 101.545,Z 87.000,A 180.000,B 0.000,C 180.000} C_DIS
LIN {X 93.321,Y 101.709,Z 87.000,A 180.000,B 0.000,C 180.000} C_DIS
LIN {X 93.335,Y 101.723,Z 87.000,A 180.000,B 0.000,C 180.000} C_DIS
LIN {X 93.500,Y 101.881,Z 87.000,A 180.000,B 0.000,C 180.000} C_DIS
LIN {X 93.524,Y 101.902,Z 87.000,A 180.000,B 0.000,C 180.000} C_DIS
LIN {X 93.679,Y 102.032,Z 87.000,A 180.000,B 0.000,C 180.000} C_DIS
LIN {X 93.737,Y 102.081,Z 87.000,A 180.000,B 0.000,C 180.000} C_DIS
LIN {X 93.857,Y 102.180,Z 87.000,A 180.000,B 0.000,C 180.000} C_DIS
LIN {X 93.960,Y 102.260,Z 87.000,A 180.000,B 0.000,C 180.000} C_DIS
LIN {X 94.036,Y 102.316,Z 87.000,A 180.000,B 0.000,C 180.000} C_DIS
LIN {X 94.215,Y 102.436,Z 87.000,A 180.000,B 0.000,C 180.000} C_DIS
LIN {X 94.394,Y 102.550,Z 87.000,A 180.000,B 0.000,C 180.000} C_DIS
LIN {X 94.501,Y 102.617,Z 87.000,A 180.000,B 0.000,C 180.000} C_DIS
LIN {X 94.573,Y 102.659,Z 87.000,A 180.000,B 0.000,C 180.000} C_DIS
LIN {X 94.751,Y 102.756,Z 87.000,A 180.000,B 0.000,C 180.000} C_DIS
LIN {X 94.832,Y 102.796,Z 87.000,A 180.000,B 0.000,C 180.000} C_DIS
LIN {X 94.930,Y 102.842,Z 87.000,A 180.000,B 0.000,C 180.000} C_DIS
LIN {X 95.109,Y 102.926,Z 87.000,A 180.000,B 0.000,C 180.000} C_DIS
LIN {X 95.217,Y 102.975,Z 87.000,A 180.000,B 0.000,C 180.000} C_DIS
LIN {X 95.288,Y 103.005,Z 87.000,A 180.000,B 0.000,C 180.000} C_DIS
LIN {X 95.466,Y 103.072,Z 87.000,A 180.000,B 0.000,C 180.000} C_DIS
LIN {X 95.645,Y 103.130,Z 87.000,A 180.000,B 0.000,C 180.000} C_DIS
LIN {X 95.717,Y 103.153,Z 87.000,A 180.000,B 0.000,C 180.000} C_DIS
LIN {X 95.824,Y 103.188,Z 87.000,A 180.000,B 0.000,C 180.000} C_DIS
LIN {X 96.003,Y 103.240,Z 87.000,A 180.000,B 0.000,C 180.000} C_DIS
LIN {X 96.181,Y 103.283,Z 87.000,A 180.000,B 0.000,C 180.000} C_DIS
LIN {X 96.360,Y 103.317,Z 87.000,A 180.000,B 0.000,C 180.000} C_DIS
LIN {X 96.539,Y 103.351,Z 87.000,A 180.000,B 0.000,C 180.000} C_DIS
LIN {X 96.718,Y 103.380,Z 87.000,A 180.000,B 0.000,C 180.000} C_DIS
LIN {X 96.897,Y 103.400,Z 87.000,A 180.000,B 0.000,C 180.000} C_DIS
LIN {X 97.075,Y 103.413,Z 87.000,A 180.000,B 0.000,C 180.000} C_DIS
LIN {X 97.254,Y 103.424,Z 87.000,A 180.000,B 0.000,C 180.000} C_DIS
LIN {X 97.433,Y 103.432,Z 87.000,A 180.000,B 0.000,C 180.000} C_DIS
LIN {X 97.612,Y 103.430,Z 87.000,A 180.000,B 0.000,C 180.000} C_DIS
LIN {X 97.790,Y 103.422,Z 87.000,A 180.000,B 0.000,C 180.000} C_DIS
LIN {X 97.969,Y 103.410,Z 87.000,A 180.000,B 0.000,C 180.000} C_DIS
LIN {X 98.148,Y 103.396,Z 87.000,A 180.000,B 0.000,C 180.000} C_DIS
LIN {X 98.327,Y 103.374,Z 87.000,A 180.000,B 0.000,C 180.000} C_DIS
LIN {X 98.505,Y 103.343,Z 87.000,A 180.000,B 0.000,C 180.000} C_DIS
LIN {X 98.684,Y 103.309,Z 87.000,A 180.000,B 0.000,C 180.000} C_DIS
LIN {X 98.863,Y 103.273,Z 87.000,A 180.000,B 0.000,C 180.000} C_DIS
LIN {X 99.042,Y 103.228,Z 87.000,A 180.000,B 0.000,C 180.000} C_DIS
LIN {X 99.221,Y 103.174,Z 87.000,A 180.000,B 0.000,C 180.000} C_DIS
LIN {X 99.399,Y 103.116,Z 87.000,A 180.000,B 0.000,C 180.000} C_DIS
LIN {X 99.578,Y 103.056,Z 87.000,A 180.000,B 0.000,C 180.000} C_DIS
LIN {X 99.757,Y 102.986,Z 87.000,A 180.000,B 0.000,C 180.000} C_DIS
LIN {X 99.783,Y 102.975,Z 87.000,A 180.000,B 0.000,C 180.000} C_DIS
LIN {X 99.936,Y 102.906,Z 87.000,A 180.000,B 0.000,C 180.000} C_DIS
LIN {X 100.114,Y 102.821,Z 87.000,A 180.000,B 0.000,C 180.000} C_DIS
LIN {X 100.168,Y 102.796,Z 87.000,A 180.000,B 0.000,C 180.000} C_DIS
LIN {X 100.293,Y 102.733,Z 87.000,A 180.000,B 0.000,C 180.000} C_DIS
LIN {X 100.472,Y 102.633,Z 87.000,A 180.000,B 0.000,C 180.000} C_DIS
LIN {X 100.499,Y 102.617,Z 87.000,A 180.000,B 0.000,C 180.000} C_DIS
LIN {X 100.651,Y 102.522,Z 87.000,A 180.000,B 0.000,C 180.000} C_DIS
LIN {X 100.782,Y 102.438,Z 87.000,A 180.000,B 0.000,C 180.000} C_DIS
LIN {X 100.829,Y 102.408,Z 87.000,A 180.000,B 0.000,C 180.000} C_DIS
LIN {X 101.008,Y 102.284,Z 87.000,A 180.000,B 0.000,C 180.000} C_DIS
LIN {X 101.040,Y 102.260,Z 87.000,A 180.000,B 0.000,C 180.000} C_DIS
LIN {X 101.187,Y 102.143,Z 87.000,A 180.000,B 0.000,C 180.000} C_DIS
LIN {X 101.366,Y 101.995,Z 87.000,A 180.000,B 0.000,C 180.000} C_DIS
LIN {X 101.476,Y 101.902,Z 87.000,A 180.000,B 0.000,C 180.000} C_DIS
LIN {X 101.545,Y 101.840,Z 87.000,A 180.000,B 0.000,C 180.000} C_DIS
LIN {X 101.665,Y 101.723,Z 87.000,A 180.000,B 0.000,C 180.000} C_DIS
LIN {X 101.723,Y 101.662,Z 87.000,A 180.000,B 0.000,C 180.000} C_DIS
LIN {X 101.834,Y 101.545,Z 87.000,A 180.000,B 0.000,C 180.000} C_DIS
LIN {X 101.902,Y 101.472,Z 87.000,A 180.000,B 0.000,C 180.000} C_DIS
LIN {X 101.999,Y 101.366,Z 87.000,A 180.000,B 0.000,C 180.000} C_DIS
LIN {X 102.081,Y 101.270,Z 87.000,A 180.000,B 0.000,C 180.000} C_DIS
LIN {X 102.147,Y 101.187,Z 87.000,A 180.000,B 0.000,C 180.000} C_DIS
LIN {X 102.260,Y 101.034,Z 87.000,A 180.000,B 0.000,C 180.000} C_DIS
LIN {X 102.279,Y 101.008,Z 87.000,A 180.000,B 0.000,C 180.000} C_DIS
LIN {X 102.408,Y 100.829,Z 87.000,A 180.000,B 0.000,C 180.000} C_DIS
LIN {X 102.438,Y 100.786,Z 87.000,A 180.000,B 0.000,C 180.000} C_DIS
LIN {X 102.527,Y 100.651,Z 87.000,A 180.000,B 0.000,C 180.000} C_DIS
LIN {X 102.617,Y 100.497,Z 87.000,A 180.000,B 0.000,C 180.000} C_DIS
LIN {X 102.631,Y 100.472,Z 87.000,A 180.000,B 0.000,C 180.000} C_DIS
LIN {X 102.729,Y 100.293,Z 87.000,A 180.000,B 0.000,C 180.000} C_DIS
LIN {X 102.796,Y 100.170,Z 87.000,A 180.000,B 0.000,C 180.000} C_DIS
LIN {X 102.825,Y 100.114,Z 87.000,A 180.000,B 0.000,C 180.000} C_DIS
LIN {X 102.909,Y 99.936,Z 87.000,A 180.000,B 0.000,C 180.000} C_DIS
LIN {X 102.975,Y 99.776,Z 87.000,A 180.000,B 0.000,C 180.000} C_DIS
LIN {X 103.053,Y 99.578,Z 87.000,A 180.000,B 0.000,C 180.000} C_DIS
LIN {X 103.120,Y 99.399,Z 87.000,A 180.000,B 0.000,C 180.000} C_DIS
LIN {X 103.153,Y 99.297,Z 87.000,A 180.000,B 0.000,C 180.000} C_DIS
LIN {X 103.177,Y 99.221,Z 87.000,A 180.000,B 0.000,C 180.000} C_DIS
LIN {X 103.224,Y 99.042,Z 87.000,A 180.000,B 0.000,C 180.000} C_DIS
LIN {X 103.270,Y 98.863,Z 87.000,A 180.000,B 0.000,C 180.000} C_DIS
LIN {X 103.313,Y 98.684,Z 87.000,A 180.000,B 0.000,C 180.000} C_DIS
LIN {X 103.332,Y 98.586,Z 87.000,A 180.000,B 0.000,C 180.000} C_DIS
LIN {X 103.346,Y 98.505,Z 87.000,A 180.000,B 0.000,C 180.000} C_DIS
LIN {X 103.371,Y 98.327,Z 87.000,A 180.000,B 0.000,C 180.000} C_DIS
LIN {X 103.393,Y 98.148,Z 87.000,A 180.000,B 0.000,C 180.000} C_DIS
LIN {X 103.413,Y 97.969,Z 87.000,A 180.000,B 0.000,C 180.000} C_DIS
LIN {X 103.425,Y 97.790,Z 87.000,A 180.000,B 0.000,C 180.000} C_DIS
LIN {X 103.428,Y 97.612,Z 87.000,A 180.000,B 0.000,C 180.000} C_DIS
LIN {X 103.428,Y 97.433,Z 87.000,A 180.000,B 0.000,C 180.000} C_DIS
LIN {X 103.426,Y 97.254,Z 87.000,A 180.000,B 0.000,C 180.000} C_DIS
LIN {X 103.417,Y 97.075,Z 87.000,A 180.000,B 0.000,C 180.000} C_DIS
LIN {X 103.399,Y 96.897,Z 87.000,A 180.000,B 0.000,C 180.000} C_DIS
LIN {X 103.376,Y 96.718,Z 87.000,A 180.000,B 0.000,C 180.000} C_DIS
LIN {X 103.353,Y 96.539,Z 87.000,A 180.000,B 0.000,C 180.000} C_DIS
LIN {X 103.332,Y 96.414,Z 87.000,A 180.000,B 0.000,C 180.000} C_DIS
LIN {X 103.322,Y 96.360,Z 87.000,A 180.000,B 0.000,C 180.000} C_DIS
LIN {X 103.281,Y 96.181,Z 87.000,A 180.000,B 0.000,C 180.000} C_DIS
LIN {X 103.236,Y 96.003,Z 87.000,A 180.000,B 0.000,C 180.000} C_DIS
LIN {X 103.189,Y 95.824,Z 87.000,A 180.000,B 0.000,C 180.000} C_DIS
LIN {X 103.153,Y 95.703,Z 87.000,A 180.000,B 0.000,C 180.000} C_DIS
LIN {X 103.135,Y 95.645,Z 87.000,A 180.000,B 0.000,C 180.000} C_DIS
LIN {X 103.070,Y 95.466,Z 87.000,A 180.000,B 0.000,C 180.000} C_DIS
LIN {X 103.000,Y 95.288,Z 87.000,A 180.000,B 0.000,C 180.000} C_DIS
LIN {X 102.975,Y 95.224,Z 87.000,A 180.000,B 0.000,C 180.000} C_DIS
LIN {X 102.928,Y 95.109,Z 87.000,A 180.000,B 0.000,C 180.000} C_DIS
LIN {X 102.847,Y 94.930,Z 87.000,A 180.000,B 0.000,C 180.000} C_DIS
LIN {X 102.796,Y 94.830,Z 87.000,A 180.000,B 0.000,C 180.000} C_DIS
LIN {X 102.754,Y 94.751,Z 87.000,A 180.000,B 0.000,C 180.000} C_DIS
LIN {X 102.656,Y 94.573,Z 87.000,A 180.000,B 0.000,C 180.000} C_DIS
LIN {X 102.617,Y 94.503,Z 87.000,A 180.000,B 0.000,C 180.000} C_DIS
LIN {X 102.554,Y 94.394,Z 87.000,A 180.000,B 0.000,C 180.000} C_DIS
LIN {X 102.439,Y 94.215,Z 87.000,A 180.000,B 0.000,C 180.000} C_DIS
LIN {X 102.438,Y 94.214,Z 87.000,A 180.000,B 0.000,C 180.000} C_DIS
LIN {X 102.311,Y 94.036,Z 87.000,A 180.000,B 0.000,C 180.000} C_DIS
LIN {X 102.260,Y 93.966,Z 87.000,A 180.000,B 0.000,C 180.000} C_DIS
LIN {X 102.180,Y 93.857,Z 87.000,A 180.000,B 0.000,C 180.000} C_DIS
LIN {X 102.081,Y 93.730,Z 87.000,A 180.000,B 0.000,C 180.000} C_DIS
LIN {X 102.037,Y 93.679,Z 87.000,A 180.000,B 0.000,C 180.000} C_DIS
LIN {X 101.902,Y 93.528,Z 87.000,A 180.000,B 0.000,C 180.000} C_DIS
LIN {X 101.875,Y 93.500,Z 87.000,A 180.000,B 0.000,C 180.000} C_DIS
LIN {X 101.723,Y 93.338,Z 87.000,A 180.000,B 0.000,C 180.000} C_DIS
LIN {X 101.707,Y 93.321,Z 87.000,A 180.000,B 0.000,C 180.000} C_DIS
LIN {X 101.545,Y 93.160,Z 87.000,A 180.000,B 0.000,C 180.000} C_DIS
LIN {X 101.525,Y 93.142,Z 87.000,A 180.000,B 0.000,C 180.000} C_DIS
LIN {X 101.366,Y 93.005,Z 87.000,A 180.000,B 0.000,C 180.000} C_DIS
LIN {X 101.187,Y 92.857,Z 87.000,A 180.000,B 0.000,C 180.000} C_DIS
LIN {X 101.099,Y 92.785,Z 87.000,A 180.000,B 0.000,C 180.000} C_DIS
LIN {X 101.008,Y 92.716,Z 87.000,A 180.000,B 0.000,C 180.000} C_DIS
LIN {X 100.850,Y 92.606,Z 87.000,A 180.000,B 0.000,C 180.000} C_DIS
LIN {X 100.829,Y 92.592,Z 87.000,A 180.000,B 0.000,C 180.000} C_DIS
LIN {X 100.651,Y 92.478,Z 87.000,A 180.000,B 0.000,C 180.000} C_DIS
LIN {X 100.570,Y 92.427,Z 87.000,A 180.000,B 0.000,C 180.000} C_DIS
LIN {X 100.472,Y 92.367,Z 87.000,A 180.000,B 0.000,C 180.000} C_DIS
LIN {X 100.293,Y 92.267,Z 87.000,A 180.000,B 0.000,C 180.000} C_DIS
LIN {X 100.258,Y 92.249,Z 87.000,A 180.000,B 0.000,C 180.000} C_DIS
LIN {X 100.114,Y 92.179,Z 87.000,A 180.000,B 0.000,C 180.000} C_DIS
LIN {X 99.936,Y 92.094,Z 87.000,A 180.000,B 0.000,C 180.000} C_DIS
LIN {X 99.883,Y 92.070,Z 87.000,A 180.000,B 0.000,C 180.000} C_DIS
LIN {X 99.757,Y 92.014,Z 87.000,A 180.000,B 0.000,C 180.000} C_DIS
LIN {X 99.578,Y 91.944,Z 87.000,A 180.000,B 0.000,C 180.000} C_DIS
LIN {X 99.420,Y 91.891,Z 87.000,A 180.000,B 0.000,C 180.000} C_DIS
LIN {X 99.221,Y 91.826,Z 87.000,A 180.000,B 0.000,C 180.000} C_DIS
LIN {X 99.042,Y 91.772,Z 87.000,A 180.000,B 0.000,C 180.000} C_DIS
LIN {X 98.863,Y 91.727,Z 87.000,A 180.000,B 0.000,C 180.000} C_DIS
LIN {X 98.792,Y 91.712,Z 87.000,A 180.000,B 0.000,C 180.000} C_DIS
LIN {X 98.684,Y 91.691,Z 87.000,A 180.000,B 0.000,C 180.000} C_DIS
LIN {X 98.505,Y 91.657,Z 87.000,A 180.000,B 0.000,C 180.000} C_DIS
LIN {X 98.327,Y 91.626,Z 87.000,A 180.000,B 0.000,C 180.000} C_DIS
LIN {X 98.148,Y 91.604,Z 87.000,A 180.000,B 0.000,C 180.000} C_DIS
LIN {X 97.969,Y 91.590,Z 87.000,A 180.000,B 0.000,C 180.000} C_DIS
LIN {X 97.790,Y 91.578,Z 87.000,A 180.000,B 0.000,C 180.000} C_DIS
LIN {X 97.612,Y 91.570,Z 87.000,A 180.000,B 0.000,C 180.000} C_DIS
LIN {X 97.433,Y 91.568,Z 87.000,A 180.000,B 0.000,C 180.000} C_DIS
LIN {X 97.254,Y 91.576,Z 87.000,A 180.000,B 0.000,C 180.000} C_DIS
LIN {X 97.075,Y 91.587,Z 87.000,A 180.000,B 0.000,C 180.000} C_DIS
LIN {X 96.897,Y 91.600,Z 87.000,A 180.000,B 0.000,C 180.000} C_DIS
LIN {X 96.718,Y 91.620,Z 87.000,A 180.000,B 0.000,C 180.000} C_DIS
LIN {X 96.539,Y 91.649,Z 87.000,A 180.000,B 0.000,C 180.000} C_DIS
LIN {X 96.360,Y 91.683,Z 87.000,A 180.000,B 0.000,C 180.000} C_DIS
LIN {X 96.208,Y 91.712,Z 87.000,A 180.000,B 0.000,C 180.000} C_DIS
LIN {X 96.181,Y 91.717,Z 87.000,A 180.000,B 0.000,C 180.000} C_DIS
LIN {X 96.003,Y 91.760,Z 87.000,A 180.000,B 0.000,C 180.000} C_DIS
LIN {X 95.824,Y 91.812,Z 87.000,A 180.000,B 0.000,C 180.000} C_DIS
LIN {X 95.645,Y 91.870,Z 87.000,A 180.000,B 0.000,C 180.000} C_DIS
LIN {X 95.580,Y 91.891,Z 87.000,A 180.000,B 0.000,C 180.000} C_DIS
LIN {X 95.466,Y 91.928,Z 87.000,A 180.000,B 0.000,C 180.000} C_DIS
LIN {X 95.288,Y 91.995,Z 87.000,A 180.000,B 0.000,C 180.000} C_DIS
LIN {X 95.117,Y 92.070,Z 87.000,A 180.000,B 0.000,C 180.000} C_DIS
LIN {X 95.109,Y 92.074,Z 87.000,A 180.000,B 0.000,C 180.000} C_DIS
LIN {X 94.930,Y 92.158,Z 87.000,A 180.000,B 0.000,C 180.000} C_DIS
LIN {X 94.751,Y 92.244,Z 87.000,A 180.000,B 0.000,C 180.000} C_DIS
LIN {X 94.742,Y 92.249,Z 87.000,A 180.000,B 0.000,C 180.000} C_DIS
LIN {X 94.573,Y 92.341,Z 87.000,A 180.000,B 0.000,C 180.000} C_DIS
LIN {X 94.430,Y 92.427,Z 87.000,A 180.000,B 0.000,C 180.000} C_DIS
LIN {X 94.215,Y 92.564,Z 87.000,A 180.000,B 0.000,C 180.000} C_DIS
LIN {X 94.150,Y 92.606,Z 87.000,A 180.000,B 0.000,C 180.000} C_DIS
LIN {X 94.036,Y 92.684,Z 87.000,A 180.000,B 0.000,C 180.000} C_DIS
LIN {X 93.901,Y 92.785,Z 87.000,A 180.000,B 0.000,C 180.000} C_DIS
LIN {X 93.857,Y 92.820,Z 87.000,A 180.000,B 0.000,C 180.000} C_DIS
LIN {X 93.679,Y 92.968,Z 87.000,A 180.000,B 0.000,C 180.000} C_DIS
LIN {X 93.500,Y 93.119,Z 87.000,A 180.000,B 0.000,C 180.000} C_DIS
LIN {X 93.475,Y 93.142,Z 87.000,A 180.000,B 0.000,C 180.000} C_DIS
LIN {X 93.321,Y 93.291,Z 87.000,A 180.000,B 0.000,C 180.000} C_DIS
LIN {X 93.293,Y 93.321,Z 87.000,A 180.000,B 0.000,C 180.000} C_DIS
LIN {X 93.142,Y 93.481,Z 87.000,A 180.000,B 0.000,C 180.000} C_DIS
LIN {X 93.125,Y 93.500,Z 87.000,A 180.000,B 0.000,C 180.000} C_DIS
LIN {X 92.964,Y 93.678,Z 87.000,A 180.000,B 0.000,C 180.000} C_DIS
LIN {X 92.963,Y 93.679,Z 87.000,A 180.000,B 0.000,C 180.000} C_DIS
LIN {X 92.820,Y 93.857,Z 87.000,A 180.000,B 0.000,C 180.000} C_DIS
LIN {X 92.785,Y 93.904,Z 87.000,A 180.000,B 0.000,C 180.000} C_DIS
LIN {X 92.689,Y 94.036,Z 87.000,A 180.000,B 0.000,C 180.000} C_DIS
LIN {X 92.606,Y 94.151,Z 87.000,A 180.000,B 0.000,C 180.000} C_DIS
LIN {X 92.561,Y 94.215,Z 87.000,A 180.000,B 0.000,C 180.000} C_DIS
LIN {X 92.446,Y 94.394,Z 87.000,A 180.000,B 0.000,C 180.000} C_DIS
LIN {X 92.427,Y 94.426,Z 87.000,A 180.000,B 0.000,C 180.000} C_DIS
LIN {X 92.344,Y 94.573,Z 87.000,A 180.000,B 0.000,C 180.000} C_DIS
LIN {X 92.246,Y 94.751,Z 87.000,A 180.000,B 0.000,C 180.000} C_DIS
LIN {X 92.153,Y 94.930,Z 87.000,A 180.000,B 0.000,C 180.000} C_DIS
LIN {X 92.072,Y 95.109,Z 87.000,A 180.000,B 0.000,C 180.000} C_DIS
LIN {X 92.070,Y 95.114,Z 87.000,A 180.000,B 0.000,C 180.000} C_DIS
LIN {X 92.000,Y 95.288,Z 87.000,A 180.000,B 0.000,C 180.000} C_DIS
LIN {X 91.930,Y 95.466,Z 87.000,A 180.000,B 0.000,C 180.000} C_DIS
LIN {X 91.891,Y 95.569,Z 87.000,A 180.000,B 0.000,C 180.000} C_DIS
LIN {X 91.865,Y 95.645,Z 87.000,A 180.000,B 0.000,C 180.000} C_DIS
LIN {X 91.811,Y 95.824,Z 87.000,A 180.000,B 0.000,C 180.000} C_DIS
LIN {X 91.764,Y 96.003,Z 87.000,A 180.000,B 0.000,C 180.000} C_DIS
LIN {X 91.719,Y 96.181,Z 87.000,A 180.000,B 0.000,C 180.000} C_DIS
LIN {X 91.712,Y 96.206,Z 87.000,A 180.000,B 0.000,C 180.000} C_DIS
LIN {X 91.678,Y 96.360,Z 87.000,A 180.000,B 0.000,C 180.000} C_DIS
LIN {X 91.647,Y 96.539,Z 87.000,A 180.000,B 0.000,C 180.000} C_DIS
LIN {X 91.624,Y 96.718,Z 87.000,A 180.000,B 0.000,C 180.000} C_DIS
LIN {X 91.607,Y 96.850,Z 87.000,A 180.000,B 0.000,C 180.000} C_DIS
LIN {X 91.601,Y 96.897,Z 87.000,A 180.000,B 0.000,C 180.000} C_DIS
LIN {X 91.583,Y 97.075,Z 87.000,A 180.000,B 0.000,C 180.000} C_DIS
LIN {X 91.574,Y 97.254,Z 87.000,A 180.000,B 0.000,C 180.000} C_DIS
LIN {X 91.572,Y 97.433,Z 87.000,A 180.000,B 0.000,C 180.000} C_DIS
LIN {X 91.572,Y 97.612,Z 87.000,A 180.000,B 0.000,C 180.000} C_DIS
LIN {X 91.575,Y 97.790,Z 87.000,A 180.000,B 0.000,C 180.000} C_DIS
LIN {X 91.587,Y 97.969,Z 87.000,A 180.000,B 0.000,C 180.000} C_DIS
LIN {X 91.607,Y 98.148,Z 87.000,A 180.000,B 0.000,C 180.000} C_DIS
LIN {X 91.616,Y 98.223,Z 87.000,A 180.000,B 0.000,C 180.000} C_DIS
; Link Move Starts
LIN {X 91.656,Y 98.518,Z 87.000,A 180.000,B 0.000,C 180.000} C_DIS
LIN {X 91.710,Y 98.788,Z 86.999,A 180.000,B 0.000,C 180.000} C_DIS
LIN {X 91.788,Y 99.091,Z 86.998,A 180.000,B 0.000,C 180.000} C_DIS
LIN {X 91.867,Y 99.365,Z 86.997,A 180.000,B 0.000,C 180.000} C_DIS
LIN {X 91.967,Y 99.634,Z 86.995,A 180.000,B 0.000,C 180.000} C_DIS
LIN {X 92.081,Y 99.920,Z 86.992,A 180.000,B 0.000,C 180.000} C_DIS
LIN {X 92.198,Y 100.168,Z 86.990,A 180.000,B 0.000,C 180.000} C_DIS
LIN {X 92.339,Y 100.430,Z 86.987,A 180.000,B 0.000,C 180.000} C_DIS
LIN {X 92.483,Y 100.680,Z 86.984,A 180.000,B 0.000,C 180.000} C_DIS
LIN {X 92.646,Y 100.921,Z 86.980,A 180.000,B 0.000,C 180.000} C_DIS
LIN {X 92.823,Y 101.166,Z 86.976,A 180.000,B 0.000,C 180.000} C_DIS
LIN {X 93.004,Y 101.390,Z 86.971,A 180.000,B 0.000,C 180.000} C_DIS
LIN {X 93.205,Y 101.608,Z 86.966,A 180.000,B 0.000,C 180.000} C_DIS
LIN {X 93.304,Y 101.715,Z 86.964,A 180.000,B 0.000,C 180.000} C_DIS
LIN {X 93.406,Y 101.818,Z 86.961,A 180.000,B 0.000,C 180.000} C_DIS
LIN {X 93.510,Y 101.915,Z 86.959,A 180.000,B 0.000,C 180.000} C_DIS
LIN {X 93.617,Y 102.008,Z 86.956,A 180.000,B 0.000,C 180.000} C_DIS
LIN {X 93.735,Y 102.107,Z 86.953,A 180.000,B 0.000,C 180.000} C_DIS
LIN {X 93.852,Y 102.206,Z 86.950,A 180.000,B 0.000,C 180.000} C_DIS
LIN {X 93.967,Y 102.296,Z 86.947,A 180.000,B 0.000,C 180.000} C_DIS
LIN {X 94.084,Y 102.382,Z 86.944,A 180.000,B 0.000,C 180.000} C_DIS
LIN {X 94.205,Y 102.463,Z 86.940,A 180.000,B 0.000,C 180.000} C_DIS
LIN {X 94.327,Y 102.542,Z 86.937,A 180.000,B 0.000,C 180.000} C_DIS
LIN {X 94.453,Y 102.624,Z 86.934,A 180.000,B 0.000,C 180.000} C_DIS
LIN {X 94.582,Y 102.702,Z 86.930,A 180.000,B 0.000,C 180.000} C_DIS
LIN {X 94.703,Y 102.770,Z 86.927,A 180.000,B 0.000,C 180.000} C_DIS
LIN {X 94.826,Y 102.833,Z 86.924,A 180.000,B 0.000,C 180.000} C_DIS
LIN {X 94.965,Y 102.900,Z 86.920,A 180.000,B 0.000,C 180.000} C_DIS
LIN {X 95.104,Y 102.967,Z 86.916,A 180.000,B 0.000,C 180.000} C_DIS
LIN {X 95.234,Y 103.027,Z 86.912,A 180.000,B 0.000,C 180.000} C_DIS
LIN {X 95.367,Y 103.081,Z 86.908,A 180.000,B 0.000,C 180.000} C_DIS
LIN {X 95.505,Y 103.132,Z 86.904,A 180.000,B 0.000,C 180.000} C_DIS
LIN {X 95.644,Y 103.179,Z 86.900,A 180.000,B 0.000,C 180.000} C_DIS
LIN {X 95.790,Y 103.228,Z 86.896,A 180.000,B 0.000,C 180.000} C_DIS
LIN {X 95.936,Y 103.275,Z 86.892,A 180.000,B 0.000,C 180.000} C_DIS
LIN {X 96.070,Y 103.311,Z 86.888,A 180.000,B 0.000,C 180.000} C_DIS
LIN {X 96.205,Y 103.342,Z 86.884,A 180.000,B 0.000,C 180.000} C_DIS
LIN {X 96.355,Y 103.374,Z 86.879,A 180.000,B 0.000,C 180.000} C_DIS
LIN {X 96.505,Y 103.404,Z 86.875,A 180.000,B 0.000,C 180.000} C_DIS
LIN {X 96.642,Y 103.431,Z 86.871,A 180.000,B 0.000,C 180.000} C_DIS
LIN {X 96.781,Y 103.452,Z 86.866,A 180.000,B 0.000,C 180.000} C_DIS
LIN {X 96.932,Y 103.468,Z 86.862,A 180.000,B 0.000,C 180.000} C_DIS
LIN {X 97.083,Y 103.481,Z 86.857,A 180.000,B 0.000,C 180.000} C_DIS
LIN {X 97.234,Y 103.492,Z 86.852,A 180.000,B 0.000,C 180.000} C_DIS
LIN {X 97.384,Y 103.502,Z 86.847,A 180.000,B 0.000,C 180.000} C_DIS
LIN {X 97.526,Y 103.506,Z 86.843,A 180.000,B 0.000,C 180.000} C_DIS
LIN {X 97.668,Y 103.504,Z 86.838,A 180.000,B 0.000,C 180.000} C_DIS
LIN {X 97.744,Y 103.501,Z 86.835,A 180.000,B 0.000,C 180.000} C_DIS
LIN {X 97.820,Y 103.498,Z 86.833,A 180.000,B 0.000,C 180.000} C_DIS
LIN {X 97.896,Y 103.494,Z 86.830,A 180.000,B 0.000,C 180.000} C_DIS
LIN {X 97.972,Y 103.491,Z 86.828,A 180.000,B 0.000,C 180.000} C_DIS
LIN {X 98.047,Y 103.487,Z 86.825,A 180.000,B 0.000,C 180.000} C_DIS
LIN {X 98.122,Y 103.482,Z 86.823,A 180.000,B 0.000,C 180.000} C_DIS
LIN {X 98.197,Y 103.476,Z 86.820,A 180.000,B 0.000,C 180.000} C_DIS
LIN {X 98.272,Y 103.468,Z 86.817,A 180.000,B 0.000,C 180.000} C_DIS
LIN {X 98.413,Y 103.449,Z 86.812,A 180.000,B 0.000,C 180.000} C_DIS
LIN {X 98.483,Y 103.437,Z 86.810,A 180.000,B 0.000,C 180.000} C_DIS
LIN {X 98.554,Y 103.425,Z 86.807,A 180.000,B 0.000,C 180.000} C_DIS
LIN {X 98.704,Y 103.399,Z 86.802,A 180.000,B 0.000,C 180.000} C_DIS
LIN {X 98.779,Y 103.386,Z 86.800,A 180.000,B 0.000,C 180.000} C_DIS
LIN {X 98.854,Y 103.372,Z 86.797,A 180.000,B 0.000,C 180.000} C_DIS
LIN {X 98.991,Y 103.342,Z 86.792,A 180.000,B 0.000,C 180.000} C_DIS
LIN {X 99.128,Y 103.307,Z 86.787,A 180.000,B 0.000,C 180.000} C_DIS
LIN {X 99.203,Y 103.285,Z 86.784,A 180.000,B 0.000,C 180.000} C_DIS
LIN {X 99.277,Y 103.262,Z 86.782,A 180.000,B 0.000,C 180.000} C_DIS
LIN {X 99.497,Y 103.195,Z 86.774,A 180.000,B 0.000,C 180.000} C_DIS
LIN {X 99.567,Y 103.173,Z 86.771,A 180.000,B 0.000,C 180.000} C_DIS
LIN {X 99.636,Y 103.149,Z 86.768,A 180.000,B 0.000,C 180.000} C_DIS
LIN {X 99.705,Y 103.124,Z 86.766,A 180.000,B 0.000,C 180.000} C_DIS
LIN {X 99.774,Y 103.099,Z 86.763,A 180.000,B 0.000,C 180.000} C_DIS
LIN {X 99.841,Y 103.071,Z 86.761,A 180.000,B 0.000,C 180.000} C_DIS
LIN {X 99.908,Y 103.043,Z 86.758,A 180.000,B 0.000,C 180.000} C_DIS
LIN {X 99.975,Y 103.013,Z 86.756,A 180.000,B 0.000,C 180.000} C_DIS
LIN {X 100.116,Y 102.949,Z 86.750,A 180.000,B 0.000,C 180.000} C_DIS
LIN {X 100.187,Y 102.918,Z 86.748,A 180.000,B 0.000,C 180.000} C_DIS
LIN {X 100.257,Y 102.885,Z 86.745,A 180.000,B 0.000,C 180.000} C_DIS
LIN {X 100.385,Y 102.822,Z 86.740,A 180.000,B 0.000,C 180.000} C_DIS
LIN {X 100.510,Y 102.754,Z 86.735,A 180.000,B 0.000,C 180.000} C_DIS
LIN {X 100.577,Y 102.716,Z 86.732,A 180.000,B 0.000,C 180.000} C_DIS
LIN {X 100.642,Y 102.676,Z 86.730,A 180.000,B 0.000,C 180.000} C_DIS
LIN {X 100.836,Y 102.558,Z 86.722,A 180.000,B 0.000,C 180.000} C_DIS
LIN {X 100.898,Y 102.519,Z 86.719,A 180.000,B 0.000,C 180.000} C_DIS
LIN {X 100.959,Y 102.480,Z 86.717,A 180.000,B 0.000,C 180.000} C_DIS
LIN {X 101.021,Y 102.440,Z 86.714,A 180.000,B 0.000,C 180.000} C_DIS
LIN {X 101.082,Y 102.397,Z 86.711,A 180.000,B 0.000,C 180.000} C_DIS
LIN {X 101.142,Y 102.353,Z 86.709,A 180.000,B 0.000,C 180.000} C_DIS
LIN {X 101.202,Y 102.308,Z 86.706,A 180.000,B 0.000,C 180.000} C_DIS
LIN {X 101.261,Y 102.262,Z 86.704,A 180.000,B 0.000,C 180.000} C_DIS
LIN {X 101.382,Y 102.165,Z 86.698,A 180.000,B 0.000,C 180.000} C_DIS
LIN {X 101.443,Y 102.116,Z 86.695,A 180.000,B 0.000,C 180.000} C_DIS
LIN {X 101.503,Y 102.067,Z 86.693,A 180.000,B 0.000,C 180.000} C_DIS
LIN {X 101.559,Y 102.021,Z 86.690,A 180.000,B 0.000,C 180.000} C_DIS
LIN {X 101.615,Y 101.973,Z 86.688,A 180.000,B 0.000,C 180.000} C_DIS
LIN {X 101.669,Y 101.924,Z 86.685,A 180.000,B 0.000,C 180.000} C_DIS
LIN {X 101.723,Y 101.875,Z 86.682,A 180.000,B 0.000,C 180.000} C_DIS
LIN {X 101.776,Y 101.823,Z 86.680,A 180.000,B 0.000,C 180.000} C_DIS
LIN {X 101.829,Y 101.769,Z 86.677,A 180.000,B 0.000,C 180.000} C_DIS
LIN {X 101.881,Y 101.716,Z 86.675,A 180.000,B 0.000,C 180.000} C_DIS
LIN {X 101.933,Y 101.662,Z 86.672,A 180.000,B 0.000,C 180.000} C_DIS
LIN {X 102.038,Y 101.554,Z 86.667,A 180.000,B 0.000,C 180.000} C_DIS
LIN {X 102.090,Y 101.500,Z 86.664,A 180.000,B 0.000,C 180.000} C_DIS
LIN {X 102.140,Y 101.444,Z 86.661,A 180.000,B 0.000,C 180.000} C_DIS
LIN {X 102.189,Y 101.388,Z 86.659,A 180.000,B 0.000,C 180.000} C_DIS
LIN {X 102.238,Y 101.331,Z 86.656,A 180.000,B 0.000,C 180.000} C_DIS
LIN {X 102.284,Y 101.273,Z 86.654,A 180.000,B 0.000,C 180.000} C_DIS
LIN {X 102.330,Y 101.214,Z 86.651,A 180.000,B 0.000,C 180.000} C_DIS
LIN {X 102.376,Y 101.153,Z 86.648,A 180.000,B 0.000,C 180.000} C_DIS
LIN {X 102.514,Y 100.970,Z 86.640,A 180.000,B 0.000,C 180.000} C_DIS
LIN {X 102.558,Y 100.910,Z 86.638,A 180.000,B 0.000,C 180.000} C_DIS
LIN {X 102.600,Y 100.849,Z 86.635,A 180.000,B 0.000,C 180.000} C_DIS
LIN {X 102.643,Y 100.788,Z 86.633,A 180.000,B 0.000,C 180.000} C_DIS
LIN {X 102.683,Y 100.726,Z 86.630,A 180.000,B 0.000,C 180.000} C_DIS
LIN {X 102.722,Y 100.662,Z 86.627,A 180.000,B 0.000,C 180.000} C_DIS
LIN {X 102.761,Y 100.599,Z 86.625,A 180.000,B 0.000,C 180.000} C_DIS
LIN {X 102.798,Y 100.534,Z 86.622,A 180.000,B 0.000,C 180.000} C_DIS
LIN {X 102.873,Y 100.403,Z 86.617,A 180.000,B 0.000,C 180.000} C_DIS
LIN {X 102.911,Y 100.336,Z 86.614,A 180.000,B 0.000,C 180.000} C_DIS
LIN {X 102.949,Y 100.268,Z 86.612,A 180.000,B 0.000,C 180.000} C_DIS
LIN {X 102.985,Y 100.200,Z 86.609,A 180.000,B 0.000,C 180.000} C_DIS
LIN {X 103.019,Y 100.136,Z 86.606,A 180.000,B 0.000,C 180.000} C_DIS
LIN {X 103.050,Y 100.071,Z 86.604,A 180.000,B 0.000,C 180.000} C_DIS
LIN {X 103.081,Y 100.005,Z 86.601,A 180.000,B 0.000,C 180.000} C_DIS
LIN {X 103.111,Y 99.939,Z 86.599,A 180.000,B 0.000,C 180.000} C_DIS
LIN {X 103.141,Y 99.868,Z 86.596,A 180.000,B 0.000,C 180.000} C_DIS
LIN {X 103.229,Y 99.654,Z 86.588,A 180.000,B 0.000,C 180.000} C_DIS
LIN {X 103.258,Y 99.585,Z 86.585,A 180.000,B 0.000,C 180.000} C_DIS
LIN {X 103.286,Y 99.515,Z 86.583,A 180.000,B 0.000,C 180.000} C_DIS
LIN {X 103.312,Y 99.444,Z 86.580,A 180.000,B 0.000,C 180.000} C_DIS
LIN {X 103.336,Y 99.373,Z 86.577,A 180.000,B 0.000,C 180.000} C_DIS
LIN {X 103.359,Y 99.302,Z 86.575,A 180.000,B 0.000,C 180.000} C_DIS
LIN {X 103.381,Y 99.231,Z 86.572,A 180.000,B 0.000,C 180.000} C_DIS
LIN {X 103.401,Y 99.159,Z 86.570,A 180.000,B 0.000,C 180.000} C_DIS
LIN {X 103.421,Y 99.087,Z 86.567,A 180.000,B 0.000,C 180.000} C_DIS
LIN {X 103.481,Y 98.869,Z 86.559,A 180.000,B 0.000,C 180.000} C_DIS
LIN {X 103.500,Y 98.795,Z 86.557,A 180.000,B 0.000,C 180.000} C_DIS
LIN {X 103.517,Y 98.721,Z 86.554,A 180.000,B 0.000,C 180.000} C_DIS
LIN {X 103.533,Y 98.647,Z 86.551,A 180.000,B 0.000,C 180.000} C_DIS
LIN {X 103.549,Y 98.572,Z 86.549,A 180.000,B 0.000,C 180.000} C_DIS
LIN {X 103.561,Y 98.497,Z 86.546,A 180.000,B 0.000,C 180.000} C_DIS
LIN {X 103.573,Y 98.422,Z 86.543,A 180.000,B 0.000,C 180.000} C_DIS
LIN {X 103.584,Y 98.346,Z 86.541,A 180.000,B 0.000,C 180.000} C_DIS
LIN {X 103.616,Y 98.121,Z 86.533,A 180.000,B 0.000,C 180.000} C_DIS
LIN {X 103.626,Y 98.047,Z 86.530,A 180.000,B 0.000,C 180.000} C_DIS
LIN {X 103.634,Y 97.973,Z 86.527,A 180.000,B 0.000,C 180.000} C_DIS
LIN {X 103.641,Y 97.899,Z 86.525,A 180.000,B 0.000,C 180.000} C_DIS
LIN {X 103.647,Y 97.824,Z 86.522,A 180.000,B 0.000,C 180.000} C_DIS
LIN {X 103.650,Y 97.748,Z 86.520,A 180.000,B 0.000,C 180.000} C_DIS
LIN {X 103.653,Y 97.673,Z 86.517,A 180.000,B 0.000,C 180.000} C_DIS
LIN {X 103.655,Y 97.598,Z 86.514,A 180.000,B 0.000,C 180.000} C_DIS
LIN {X 103.659,Y 97.364,Z 86.506,A 180.000,B 0.000,C 180.000} C_DIS
LIN {X 103.659,Y 97.286,Z 86.503,A 180.000,B 0.000,C 180.000} C_DIS
LIN {X 103.658,Y 97.211,Z 86.501,A 180.000,B 0.000,C 180.000} C_DIS
LIN {X 103.656,Y 97.137,Z 86.498,A 180.000,B 0.000,C 180.000} C_DIS
LIN {X 103.652,Y 97.063,Z 86.496,A 180.000,B 0.000,C 180.000} C_DIS
LIN {X 103.647,Y 96.989,Z 86.493,A 180.000,B 0.000,C 180.000} C_DIS
LIN {X 103.640,Y 96.913,Z 86.490,A 180.000,B 0.000,C 180.000} C_DIS
LIN {X 103.632,Y 96.837,Z 86.488,A 180.000,B 0.000,C 180.000} C_DIS
LIN {X 103.607,Y 96.610,Z 86.480,A 180.000,B 0.000,C 180.000} C_DIS
LIN {X 103.598,Y 96.535,Z 86.477,A 180.000,B 0.000,C 180.000} C_DIS
LIN {X 103.589,Y 96.461,Z 86.474,A 180.000,B 0.000,C 180.000} C_DIS
LIN {X 103.578,Y 96.387,Z 86.472,A 180.000,B 0.000,C 180.000} C_DIS
LIN {X 103.564,Y 96.312,Z 86.469,A 180.000,B 0.000,C 180.000} C_DIS
LIN {X 103.550,Y 96.237,Z 86.466,A 180.000,B 0.000,C 180.000} C_DIS
LIN {X 103.534,Y 96.162,Z 86.464,A 180.000,B 0.000,C 180.000} C_DIS
LIN {X 103.517,Y 96.088,Z 86.461,A 180.000,B 0.000,C 180.000} C_DIS
LIN {X 103.463,Y 95.861,Z 86.453,A 180.000,B 0.000,C 180.000} C_DIS
LIN {X 103.444,Y 95.785,Z 86.450,A 180.000,B 0.000,C 180.000} C_DIS
LIN {X 103.426,Y 95.714,Z 86.448,A 180.000,B 0.000,C 180.000} C_DIS
LIN {X 103.406,Y 95.642,Z 86.445,A 180.000,B 0.000,C 180.000} C_DIS
LIN {X 103.384,Y 95.572,Z 86.443,A 180.000,B 0.000,C 180.000} C_DIS
LIN {X 103.362,Y 95.501,Z 86.440,A 180.000,B 0.000,C 180.000} C_DIS
LIN {X 103.336,Y 95.428,Z 86.437,A 180.000,B 0.000,C 180.000} C_DIS
LIN {X 103.310,Y 95.355,Z 86.435,A 180.000,B 0.000,C 180.000} C_DIS
LIN {X 103.283,Y 95.282,Z 86.432,A 180.000,B 0.000,C 180.000} C_DIS
LIN {X 103.202,Y 95.067,Z 86.424,A 180.000,B 0.000,C 180.000} C_DIS
LIN {X 103.173,Y 94.996,Z 86.421,A 180.000,B 0.000,C 180.000} C_DIS
LIN {X 103.144,Y 94.926,Z 86.418,A 180.000,B 0.000,C 180.000} C_DIS
LIN {X 103.114,Y 94.857,Z 86.416,A 180.000,B 0.000,C 180.000} C_DIS
LIN {X 103.082,Y 94.788,Z 86.413,A 180.000,B 0.000,C 180.000} C_DIS
LIN {X 103.049,Y 94.721,Z 86.411,A 180.000,B 0.000,C 180.000} C_DIS
LIN {X 103.015,Y 94.653,Z 86.408,A 180.000,B 0.000,C 180.000} C_DIS
LIN {X 102.979,Y 94.584,Z 86.405,A 180.000,B 0.000,C 180.000} C_DIS
LIN {X 102.906,Y 94.446,Z 86.400,A 180.000,B 0.000,C 180.000} C_DIS
LIN {X 102.869,Y 94.377,Z 86.397,A 180.000,B 0.000,C 180.000} C_DIS
LIN {X 102.833,Y 94.311,Z 86.394,A 180.000,B 0.000,C 180.000} C_DIS
LIN {X 102.796,Y 94.246,Z 86.392,A 180.000,B 0.000,C 180.000} C_DIS
LIN {X 102.758,Y 94.181,Z 86.389,A 180.000,B 0.000,C 180.000} C_DIS
LIN {X 102.718,Y 94.118,Z 86.387,A 180.000,B 0.000,C 180.000} C_DIS
LIN {X 102.676,Y 94.053,Z 86.384,A 180.000,B 0.000,C 180.000} C_DIS
LIN {X 102.633,Y 93.989,Z 86.381,A 180.000,B 0.000,C 180.000} C_DIS
LIN {X 102.589,Y 93.926,Z 86.378,A 180.000,B 0.000,C 180.000} C_DIS
LIN {X 102.500,Y 93.799,Z 86.373,A 180.000,B 0.000,C 180.000} C_DIS
LIN {X 102.455,Y 93.735,Z 86.370,A 180.000,B 0.000,C 180.000} C_DIS
LIN {X 102.409,Y 93.672,Z 86.368,A 180.000,B 0.000,C 180.000} C_DIS
LIN {X 102.363,Y 93.609,Z 86.365,A 180.000,B 0.000,C 180.000} C_DIS
LIN {X 102.317,Y 93.550,Z 86.362,A 180.000,B 0.000,C 180.000} C_DIS
LIN {X 102.270,Y 93.492,Z 86.360,A 180.000,B 0.000,C 180.000} C_DIS
LIN {X 102.222,Y 93.434,Z 86.357,A 180.000,B 0.000,C 180.000} C_DIS
LIN {X 102.173,Y 93.378,Z 86.354,A 180.000,B 0.000,C 180.000} C_DIS
LIN {X 102.121,Y 93.320,Z 86.352,A 180.000,B 0.000,C 180.000} C_DIS
LIN {X 102.016,Y 93.204,Z 86.346,A 180.000,B 0.000,C 180.000} C_DIS
LIN {X 101.963,Y 93.147,Z 86.344,A 180.000,B 0.000,C 180.000} C_DIS
LIN {X 101.912,Y 93.090,Z 86.341,A 180.000,B 0.000,C 180.000} C_DIS
LIN {X 101.859,Y 93.035,Z 86.338,A 180.000,B 0.000,C 180.000} C_DIS
LIN {X 101.805,Y 92.980,Z 86.336,A 180.000,B 0.000,C 180.000} C_DIS
LIN {X 101.751,Y 92.927,Z 86.333,A 180.000,B 0.000,C 180.000} C_DIS
LIN {X 101.695,Y 92.874,Z 86.330,A 180.000,B 0.000,C 180.000} C_DIS
LIN {X 101.638,Y 92.824,Z 86.328,A 180.000,B 0.000,C 180.000} C_DIS
LIN {X 101.580,Y 92.773,Z 86.325,A 180.000,B 0.000,C 180.000} C_DIS
LIN {X 101.522,Y 92.723,Z 86.322,A 180.000,B 0.000,C 180.000} C_DIS
LIN {X 101.404,Y 92.623,Z 86.317,A 180.000,B 0.000,C 180.000} C_DIS
LIN {X 101.346,Y 92.573,Z 86.314,A 180.000,B 0.000,C 180.000} C_DIS
LIN {X 101.286,Y 92.524,Z 86.311,A 180.000,B 0.000,C 180.000} C_DIS
LIN {X 101.226,Y 92.477,Z 86.309,A 180.000,B 0.000,C 180.000} C_DIS
LIN {X 101.166,Y 92.430,Z 86.306,A 180.000,B 0.000,C 180.000} C_DIS
LIN {X 101.104,Y 92.386,Z 86.303,A 180.000,B 0.000,C 180.000} C_DIS
LIN {X 101.042,Y 92.342,Z 86.301,A 180.000,B 0.000,C 180.000} C_DIS
LIN {X 100.977,Y 92.298,Z 86.298,A 180.000,B 0.000,C 180.000} C_DIS
LIN {X 100.912,Y 92.255,Z 86.295,A 180.000,B 0.000,C 180.000} C_DIS
LIN {X 100.781,Y 92.169,Z 86.290,A 180.000,B 0.000,C 180.000} C_DIS
LIN {X 100.717,Y 92.127,Z 86.287,A 180.000,B 0.000,C 180.000} C_DIS
LIN {X 100.652,Y 92.086,Z 86.284,A 180.000,B 0.000,C 180.000} C_DIS
LIN {X 100.586,Y 92.046,Z 86.282,A 180.000,B 0.000,C 180.000} C_DIS
LIN {X 100.520,Y 92.007,Z 86.279,A 180.000,B 0.000,C 180.000} C_DIS
LIN {X 100.453,Y 91.970,Z 86.276,A 180.000,B 0.000,C 180.000} C_DIS
LIN {X 100.385,Y 91.933,Z 86.274,A 180.000,B 0.000,C 180.000} C_DIS
LIN {X 100.316,Y 91.898,Z 86.271,A 180.000,B 0.000,C 180.000} C_DIS
LIN {X 100.247,Y 91.864,Z 86.268,A 180.000,B 0.000,C 180.000} C_DIS
LIN {X 100.108,Y 91.795,Z 86.263,A 180.000,B 0.000,C 180.000} C_DIS
LIN {X 100.038,Y 91.761,Z 86.260,A 180.000,B 0.000,C 180.000} C_DIS
LIN {X 99.967,Y 91.728,Z 86.258,A 180.000,B 0.000,C 180.000} C_DIS
LIN {X 99.898,Y 91.696,Z 86.255,A 180.000,B 0.000,C 180.000} C_DIS
LIN {X 99.828,Y 91.666,Z 86.252,A 180.000,B 0.000,C 180.000} C_DIS
LIN {X 99.758,Y 91.638,Z 86.250,A 180.000,B 0.000,C 180.000} C_DIS
LIN {X 99.687,Y 91.610,Z 86.247,A 180.000,B 0.000,C 180.000} C_DIS
LIN {X 99.613,Y 91.583,Z 86.244,A 180.000,B 0.000,C 180.000} C_DIS
LIN {X 99.539,Y 91.558,Z 86.241,A 180.000,B 0.000,C 180.000} C_DIS
LIN {X 99.391,Y 91.507,Z 86.236,A 180.000,B 0.000,C 180.000} C_DIS
LIN {X 99.318,Y 91.482,Z 86.233,A 180.000,B 0.000,C 180.000} C_DIS
LIN {X 99.245,Y 91.457,Z 86.231,A 180.000,B 0.000,C 180.000} C_DIS
LIN {X 99.171,Y 91.434,Z 86.228,A 180.000,B 0.000,C 180.000} C_DIS
LIN {X 99.097,Y 91.413,Z 86.225,A 180.000,B 0.000,C 180.000} C_DIS
LIN {X 99.023,Y 91.392,Z 86.222,A 180.000,B 0.000,C 180.000} C_DIS
LIN {X 98.948,Y 91.373,Z 86.220,A 180.000,B 0.000,C 180.000} C_DIS
LIN {X 98.873,Y 91.356,Z 86.217,A 180.000,B 0.000,C 180.000} C_DIS
LIN {X 98.798,Y 91.340,Z 86.214,A 180.000,B 0.000,C 180.000} C_DIS
LIN {X 98.721,Y 91.324,Z 86.212,A 180.000,B 0.000,C 180.000} C_DIS
LIN {X 98.567,Y 91.292,Z 86.206,A 180.000,B 0.000,C 180.000} C_DIS
LIN {X 98.490,Y 91.276,Z 86.203,A 180.000,B 0.000,C 180.000} C_DIS
LIN {X 98.414,Y 91.262,Z 86.201,A 180.000,B 0.000,C 180.000} C_DIS
LIN {X 98.338,Y 91.250,Z 86.198,A 180.000,B 0.000,C 180.000} C_DIS
LIN {X 98.262,Y 91.238,Z 86.195,A 180.000,B 0.000,C 180.000} C_DIS
LIN {X 98.185,Y 91.229,Z 86.193,A 180.000,B 0.000,C 180.000} C_DIS
LIN {X 98.108,Y 91.221,Z 86.190,A 180.000,B 0.000,C 180.000} C_DIS
LIN {X 98.031,Y 91.214,Z 86.187,A 180.000,B 0.000,C 180.000} C_DIS
LIN {X 97.953,Y 91.208,Z 86.185,A 180.000,B 0.000,C 180.000} C_DIS
LIN {X 97.876,Y 91.201,Z 86.182,A 180.000,B 0.000,C 180.000} C_DIS
LIN {X 97.798,Y 91.195,Z 86.179,A 180.000,B 0.000,C 180.000} C_DIS
LIN {X 97.721,Y 91.189,Z 86.177,A 180.000,B 0.000,C 180.000} C_DIS
LIN {X 97.643,Y 91.185,Z 86.174,A 180.000,B 0.000,C 180.000} C_DIS
LIN {X 97.566,Y 91.182,Z 86.172,A 180.000,B 0.000,C 180.000} C_DIS
LIN {X 97.488,Y 91.180,Z 86.169,A 180.000,B 0.000,C 180.000} C_DIS
LIN {X 97.411,Y 91.180,Z 86.166,A 180.000,B 0.000,C 180.000} C_DIS
LIN {X 97.333,Y 91.181,Z 86.164,A 180.000,B 0.000,C 180.000} C_DIS
LIN {X 97.256,Y 91.183,Z 86.161,A 180.000,B 0.000,C 180.000} C_DIS
LIN {X 97.177,Y 91.187,Z 86.159,A 180.000,B 0.000,C 180.000} C_DIS
LIN {X 97.099,Y 91.191,Z 86.156,A 180.000,B 0.000,C 180.000} C_DIS
LIN {X 97.020,Y 91.195,Z 86.154,A 180.000,B 0.000,C 180.000} C_DIS
LIN {X 96.942,Y 91.199,Z 86.151,A 180.000,B 0.000,C 180.000} C_DIS
LIN {X 96.787,Y 91.210,Z 86.146,A 180.000,B 0.000,C 180.000} C_DIS
LIN {X 96.633,Y 91.227,Z 86.141,A 180.000,B 0.000,C 180.000} C_DIS
LIN {X 96.479,Y 91.250,Z 86.137,A 180.000,B 0.000,C 180.000} C_DIS
LIN {X 96.325,Y 91.277,Z 86.132,A 180.000,B 0.000,C 180.000} C_DIS
LIN {X 96.171,Y 91.304,Z 86.127,A 180.000,B 0.000,C 180.000} C_DIS
LIN {X 96.018,Y 91.334,Z 86.122,A 180.000,B 0.000,C 180.000} C_DIS
LIN {X 95.867,Y 91.370,Z 86.118,A 180.000,B 0.000,C 180.000} C_DIS
LIN {X 95.717,Y 91.412,Z 86.114,A 180.000,B 0.000,C 180.000} C_DIS
LIN {X 95.567,Y 91.458,Z 86.109,A 180.000,B 0.000,C 180.000} C_DIS
LIN {X 95.417,Y 91.505,Z 86.105,A 180.000,B 0.000,C 180.000} C_DIS
LIN {X 95.269,Y 91.553,Z 86.100,A 180.000,B 0.000,C 180.000} C_DIS
LIN {X 95.123,Y 91.608,Z 86.096,A 180.000,B 0.000,C 180.000} C_DIS
LIN {X 94.978,Y 91.668,Z 86.092,A 180.000,B 0.000,C 180.000} C_DIS
LIN {X 94.835,Y 91.732,Z 86.088,A 180.000,B 0.000,C 180.000} C_DIS
LIN {X 94.693,Y 91.797,Z 86.084,A 180.000,B 0.000,C 180.000} C_DIS
LIN {X 94.551,Y 91.865,Z 86.080,A 180.000,B 0.000,C 180.000} C_DIS
LIN {X 94.412,Y 91.936,Z 86.076,A 180.000,B 0.000,C 180.000} C_DIS
LIN {X 94.276,Y 92.014,Z 86.073,A 180.000,B 0.000,C 180.000} C_DIS
LIN {X 94.142,Y 92.095,Z 86.069,A 180.000,B 0.000,C 180.000} C_DIS
LIN {X 94.009,Y 92.178,Z 86.065,A 180.000,B 0.000,C 180.000} C_DIS
LIN {X 93.877,Y 92.262,Z 86.062,A 180.000,B 0.000,C 180.000} C_DIS
LIN {X 93.747,Y 92.351,Z 86.058,A 180.000,B 0.000,C 180.000} C_DIS
LIN {X 93.622,Y 92.444,Z 86.055,A 180.000,B 0.000,C 180.000} C_DIS
LIN {X 93.499,Y 92.542,Z 86.052,A 180.000,B 0.000,C 180.000} C_DIS
LIN {X 93.377,Y 92.641,Z 86.049,A 180.000,B 0.000,C 180.000} C_DIS
LIN {X 93.256,Y 92.741,Z 86.046,A 180.000,B 0.000,C 180.000} C_DIS
LIN {X 93.139,Y 92.846,Z 86.043,A 180.000,B 0.000,C 180.000} C_DIS
LIN {X 93.025,Y 92.954,Z 86.040,A 180.000,B 0.000,C 180.000} C_DIS
LIN {X 92.915,Y 93.066,Z 86.037,A 180.000,B 0.000,C 180.000} C_DIS
LIN {X 92.807,Y 93.180,Z 86.034,A 180.000,B 0.000,C 180.000} C_DIS
LIN {X 92.699,Y 93.294,Z 86.032,A 180.000,B 0.000,C 180.000} C_DIS
LIN {X 92.595,Y 93.412,Z 86.029,A 180.000,B 0.000,C 180.000} C_DIS
LIN {X 92.401,Y 93.659,Z 86.024,A 180.000,B 0.000,C 180.000} C_DIS
LIN {X 92.214,Y 93.912,Z 86.020,A 180.000,B 0.000,C 180.000} C_DIS
LIN {X 92.042,Y 94.176,Z 86.016,A 180.000,B 0.000,C 180.000} C_DIS
LIN {X 91.887,Y 94.449,Z 86.012,A 180.000,B 0.000,C 180.000} C_DIS
LIN {X 91.738,Y 94.727,Z 86.009,A 180.000,B 0.000,C 180.000} C_DIS
LIN {X 91.610,Y 95.014,Z 86.007,A 180.000,B 0.000,C 180.000} C_DIS
LIN {X 91.494,Y 95.307,Z 86.004,A 180.000,B 0.000,C 180.000} C_DIS
LIN {X 91.390,Y 95.604,Z 86.003,A 180.000,B 0.000,C 180.000} C_DIS
LIN {X 91.308,Y 95.908,Z 86.001,A 180.000,B 0.000,C 180.000} C_DIS
LIN {X 91.233,Y 96.214,Z 86.000,A 180.000,B 0.000,C 180.000} C_DIS
LIN {X 91.179,Y 96.524,Z 86.000,A 180.000,B 0.000,C 180.000} C_DIS
LIN {X 91.168,Y 96.604,Z 86.000,A 180.000,B 0.000,C 180.000} C_DIS
; Cutting Move Starts
LIN {X 91.153,Y 96.718,Z 86.000,A 180.000,B 0.000,C 180.000} C_DIS
LIN {X 91.131,Y 96.897,Z 86.000,A 180.000,B 0.000,C 180.000} C_DIS
LIN {X 91.115,Y 97.075,Z 86.000,A 180.000,B 0.000,C 180.000} C_DIS
LIN {X 91.107,Y 97.254,Z 86.000,A 180.000,B 0.000,C 180.000} C_DIS
LIN {X 91.105,Y 97.433,Z 86.000,A 180.000,B 0.000,C 180.000} C_DIS
LIN {X 91.105,Y 97.612,Z 86.000,A 180.000,B 0.000,C 180.000} C_DIS
LIN {X 91.109,Y 97.790,Z 86.000,A 180.000,B 0.000,C 180.000} C_DIS
LIN {X 91.119,Y 97.969,Z 86.000,A 180.000,B 0.000,C 180.000} C_DIS
LIN {X 91.137,Y 98.148,Z 86.000,A 180.000,B 0.000,C 180.000} C_DIS
LIN {X 91.153,Y 98.281,Z 86.000,A 180.000,B 0.000,C 180.000} C_DIS
LIN {X 91.159,Y 98.327,Z 86.000,A 180.000,B 0.000,C 180.000} C_DIS
LIN {X 91.176,Y 98.457,Z 86.000,A 180.000,B 0.000,C 180.000} C_DIS
LIN {X 91.183,Y 98.505,Z 86.000,A 180.000,B 0.000,C 180.000} C_DIS
LIN {X 91.212,Y 98.684,Z 86.000,A 180.000,B 0.000,C 180.000} C_DIS
LIN {X 91.249,Y 98.863,Z 86.000,A 180.000,B 0.000,C 180.000} C_DIS
LIN {X 91.294,Y 99.042,Z 86.000,A 180.000,B 0.000,C 180.000} C_DIS
LIN {X 91.340,Y 99.221,Z 86.000,A 180.000,B 0.000,C 180.000} C_DIS
LIN {X 91.355,Y 99.276,Z 86.000,A 180.000,B 0.000,C 180.000} C_DIS
LIN {X 91.390,Y 99.399,Z 86.000,A 180.000,B 0.000,C 180.000} C_DIS
LIN {X 91.448,Y 99.578,Z 86.000,A 180.000,B 0.000,C 180.000} C_DIS
LIN {X 91.516,Y 99.757,Z 86.000,A 180.000,B 0.000,C 180.000} C_DIS
LIN {X 91.587,Y 99.936,Z 86.000,A 180.000,B 0.000,C 180.000} C_DIS
LIN {X 91.661,Y 100.114,Z 86.000,A 180.000,B 0.000,C 180.000} C_DIS
LIN {X 91.712,Y 100.229,Z 86.000,A 180.000,B 0.000,C 180.000} C_DIS
LIN {X 91.743,Y 100.293,Z 86.000,A 180.000,B 0.000,C 180.000} C_DIS
LIN {X 91.837,Y 100.472,Z 86.000,A 180.000,B 0.000,C 180.000} C_DIS
LIN {X 91.935,Y 100.651,Z 86.000,A 180.000,B 0.000,C 180.000} C_DIS
LIN {X 92.037,Y 100.829,Z 86.000,A 180.000,B 0.000,C 180.000} C_DIS
LIN {X 92.070,Y 100.885,Z 86.000,A 180.000,B 0.000,C 180.000} C_DIS
LIN {X 92.150,Y 101.008,Z 86.000,A 180.000,B 0.000,C 180.000} C_DIS
LIN {X 92.249,Y 101.151,Z 86.000,A 180.000,B 0.000,C 180.000} C_DIS
LIN {X 92.275,Y 101.187,Z 86.000,A 180.000,B 0.000,C 180.000} C_DIS
LIN {X 92.405,Y 101.366,Z 86.000,A 180.000,B 0.000,C 180.000} C_DIS
LIN {X 92.427,Y 101.396,Z 86.000,A 180.000,B 0.000,C 180.000} C_DIS
LIN {X 92.542,Y 101.545,Z 86.000,A 180.000,B 0.000,C 180.000} C_DIS
LIN {X 92.606,Y 101.621,Z 86.000,A 180.000,B 0.000,C 180.000} C_DIS
LIN {X 92.695,Y 101.723,Z 86.000,A 180.000,B 0.000,C 180.000} C_DIS
LIN {X 92.785,Y 101.820,Z 86.000,A 180.000,B 0.000,C 180.000} C_DIS
LIN {X 92.862,Y 101.902,Z 86.000,A 180.000,B 0.000,C 180.000} C_DIS
LIN {X 92.964,Y 102.009,Z 86.000,A 180.000,B 0.000,C 180.000} C_DIS
LIN {X 93.033,Y 102.081,Z 86.000,A 180.000,B 0.000,C 180.000} C_DIS
LIN {X 93.142,Y 102.185,Z 86.000,A 180.000,B 0.000,C 180.000} C_DIS
LIN {X 93.224,Y 102.260,Z 86.000,A 180.000,B 0.000,C 180.000} C_DIS
LIN {X 93.321,Y 102.342,Z 86.000,A 180.000,B 0.000,C 180.000} C_DIS
LIN {X 93.438,Y 102.438,Z 86.000,A 180.000,B 0.000,C 180.000} C_DIS
LIN {X 93.500,Y 102.490,Z 86.000,A 180.000,B 0.000,C 180.000} C_DIS
LIN {X 93.660,Y 102.617,Z 86.000,A 180.000,B 0.000,C 180.000} C_DIS
LIN {X 93.679,Y 102.631,Z 86.000,A 180.000,B 0.000,C 180.000} C_DIS
LIN {X 93.857,Y 102.759,Z 86.000,A 180.000,B 0.000,C 180.000} C_DIS
LIN {X 93.912,Y 102.796,Z 86.000,A 180.000,B 0.000,C 180.000} C_DIS
LIN {X 94.036,Y 102.875,Z 86.000,A 180.000,B 0.000,C 180.000} C_DIS
LIN {X 94.193,Y 102.975,Z 86.000,A 180.000,B 0.000,C 180.000} C_DIS
LIN {X 94.215,Y 102.989,Z 86.000,A 180.000,B 0.000,C 180.000} C_DIS
LIN {X 94.394,Y 103.094,Z 86.000,A 180.000,B 0.000,C 180.000} C_DIS
LIN {X 94.505,Y 103.153,Z 86.000,A 180.000,B 0.000,C 180.000} C_DIS
LIN {X 94.573,Y 103.188,Z 86.000,A 180.000,B 0.000,C 180.000} C_DIS
LIN {X 94.751,Y 103.274,Z 86.000,A 180.000,B 0.000,C 180.000} C_DIS
LIN {X 94.876,Y 103.332,Z 86.000,A 180.000,B 0.000,C 180.000} C_DIS
LIN {X 94.930,Y 103.357,Z 86.000,A 180.000,B 0.000,C 180.000} C_DIS
LIN {X 95.109,Y 103.435,Z 86.000,A 180.000,B 0.000,C 180.000} C_DIS
LIN {X 95.288,Y 103.503,Z 86.000,A 180.000,B 0.000,C 180.000} C_DIS
LIN {X 95.310,Y 103.511,Z 86.000,A 180.000,B 0.000,C 180.000} C_DIS
LIN {X 95.466,Y 103.563,Z 86.000,A 180.000,B 0.000,C 180.000} C_DIS
LIN {X 95.645,Y 103.620,Z 86.000,A 180.000,B 0.000,C 180.000} C_DIS
LIN {X 95.824,Y 103.675,Z 86.000,A 180.000,B 0.000,C 180.000} C_DIS
LIN {X 95.880,Y 103.690,Z 86.000,A 180.000,B 0.000,C 180.000} C_DIS
LIN {X 96.003,Y 103.721,Z 86.000,A 180.000,B 0.000,C 180.000} C_DIS
LIN {X 96.181,Y 103.758,Z 86.000,A 180.000,B 0.000,C 180.000} C_DIS
LIN {X 96.360,Y 103.792,Z 86.000,A 180.000,B 0.000,C 180.000} C_DIS
LIN {X 96.539,Y 103.825,Z 86.000,A 180.000,B 0.000,C 180.000} C_DIS
LIN {X 96.718,Y 103.851,Z 86.000,A 180.000,B 0.000,C 180.000} C_DIS
LIN {X 96.897,Y 103.868,Z 86.000,A 180.000,B 0.000,C 180.000} C_DIS
LIN {X 96.901,Y 103.869,Z 86.000,A 180.000,B 0.000,C 180.000} C_DIS
LIN {X 97.075,Y 103.881,Z 86.000,A 180.000,B 0.000,C 180.000} C_DIS
LIN {X 97.254,Y 103.892,Z 86.000,A 180.000,B 0.000,C 180.000} C_DIS
LIN {X 97.433,Y 103.898,Z 86.000,A 180.000,B 0.000,C 180.000} C_DIS
LIN {X 97.612,Y 103.897,Z 86.000,A 180.000,B 0.000,C 180.000} C_DIS
LIN {X 97.790,Y 103.889,Z 86.000,A 180.000,B 0.000,C 180.000} C_DIS
LIN {X 97.969,Y 103.878,Z 86.000,A 180.000,B 0.000,C 180.000} C_DIS
LIN {X 98.099,Y 103.869,Z 86.000,A 180.000,B 0.000,C 180.000} C_DIS
LIN {X 98.148,Y 103.864,Z 86.000,A 180.000,B 0.000,C 180.000} C_DIS
LIN {X 98.327,Y 103.845,Z 86.000,A 180.000,B 0.000,C 180.000} C_DIS
LIN {X 98.505,Y 103.818,Z 86.000,A 180.000,B 0.000,C 180.000} C_DIS
LIN {X 98.684,Y 103.784,Z 86.000,A 180.000,B 0.000,C 180.000} C_DIS
LIN {X 98.863,Y 103.749,Z 86.000,A 180.000,B 0.000,C 180.000} C_DIS
LIN {X 99.042,Y 103.710,Z 86.000,A 180.000,B 0.000,C 180.000} C_DIS
LIN {X 99.120,Y 103.690,Z 86.000,A 180.000,B 0.000,C 180.000} C_DIS
LIN {X 99.221,Y 103.663,Z 86.000,A 180.000,B 0.000,C 180.000} C_DIS
LIN {X 99.399,Y 103.606,Z 86.000,A 180.000,B 0.000,C 180.000} C_DIS
LIN {X 99.578,Y 103.548,Z 86.000,A 180.000,B 0.000,C 180.000} C_DIS
LIN {X 99.690,Y 103.511,Z 86.000,A 180.000,B 0.000,C 180.000} C_DIS
LIN {X 99.757,Y 103.487,Z 86.000,A 180.000,B 0.000,C 180.000} C_DIS
LIN {X 99.936,Y 103.417,Z 86.000,A 180.000,B 0.000,C 180.000} C_DIS
LIN {X 100.114,Y 103.337,Z 86.000,A 180.000,B 0.000,C 180.000} C_DIS
LIN {X 100.293,Y 103.253,Z 86.000,A 180.000,B 0.000,C 180.000} C_DIS
LIN {X 100.472,Y 103.165,Z 86.000,A 180.000,B 0.000,C 180.000} C_DIS
LIN {X 100.495,Y 103.153,Z 86.000,A 180.000,B 0.000,C 180.000} C_DIS
LIN {X 100.651,Y 103.069,Z 86.000,A 180.000,B 0.000,C 180.000} C_DIS
LIN {X 100.807,Y 102.975,Z 86.000,A 180.000,B 0.000,C 180.000} C_DIS
LIN {X 101.008,Y 102.847,Z 86.000,A 180.000,B 0.000,C 180.000} C_DIS
LIN {X 101.088,Y 102.796,Z 86.000,A 180.000,B 0.000,C 180.000} C_DIS
LIN {X 101.187,Y 102.729,Z 86.000,A 180.000,B 0.000,C 180.000} C_DIS
LIN {X 101.340,Y 102.617,Z 86.000,A 180.000,B 0.000,C 180.000} C_DIS
LIN {X 101.366,Y 102.598,Z 86.000,A 180.000,B 0.000,C 180.000} C_DIS
LIN {X 101.545,Y 102.453,Z 86.000,A 180.000,B 0.000,C 180.000} C_DIS
LIN {X 101.562,Y 102.438,Z 86.000,A 180.000,B 0.000,C 180.000} C_DIS
LIN {X 101.723,Y 102.304,Z 86.000,A 180.000,B 0.000,C 180.000} C_DIS
LIN {X 101.776,Y 102.260,Z 86.000,A 180.000,B 0.000,C 180.000} C_DIS
LIN {X 101.902,Y 102.143,Z 86.000,A 180.000,B 0.000,C 180.000} C_DIS
LIN {X 101.967,Y 102.081,Z 86.000,A 180.000,B 0.000,C 180.000} C_DIS
LIN {X 102.081,Y 101.962,Z 86.000,A 180.000,B 0.000,C 180.000} C_DIS
LIN {X 102.138,Y 101.902,Z 86.000,A 180.000,B 0.000,C 180.000} C_DIS
LIN {X 102.260,Y 101.772,Z 86.000,A 180.000,B 0.000,C 180.000} C_DIS
LIN {X 102.305,Y 101.723,Z 86.000,A 180.000,B 0.000,C 180.000} C_DIS
LIN {X 102.438,Y 101.569,Z 86.000,A 180.000,B 0.000,C 180.000} C_DIS
LIN {X 102.458,Y 101.545,Z 86.000,A 180.000,B 0.000,C 180.000} C_DIS
LIN {X 102.595,Y 101.366,Z 86.000,A 180.000,B 0.000,C 180.000} C_DIS
LIN {X 102.617,Y 101.336,Z 86.000,A 180.000,B 0.000,C 180.000} C_DIS
LIN {X 102.725,Y 101.187,Z 86.000,A 180.000,B 0.000,C 180.000} C_DIS
LIN {X 102.796,Y 101.089,Z 86.000,A 180.000,B 0.000,C 180.000} C_DIS
LIN {X 102.850,Y 101.008,Z 86.000,A 180.000,B 0.000,C 180.000} C_DIS
LIN {X 102.963,Y 100.829,Z 86.000,A 180.000,B 0.000,C 180.000} C_DIS
LIN {X 102.975,Y 100.810,Z 86.000,A 180.000,B 0.000,C 180.000} C_DIS
LIN {X 103.065,Y 100.651,Z 86.000,A 180.000,B 0.000,C 180.000} C_DIS
LIN {X 103.163,Y 100.472,Z 86.000,A 180.000,B 0.000,C 180.000} C_DIS
LIN {X 103.257,Y 100.293,Z 86.000,A 180.000,B 0.000,C 180.000} C_DIS
LIN {X 103.332,Y 100.130,Z 86.000,A 180.000,B 0.000,C 180.000} C_DIS
LIN {X 103.339,Y 100.114,Z 86.000,A 180.000,B 0.000,C 180.000} C_DIS
LIN {X 103.413,Y 99.936,Z 86.000,A 180.000,B 0.000,C 180.000} C_DIS
LIN {X 103.484,Y 99.757,Z 86.000,A 180.000,B 0.000,C 180.000} C_DIS
LIN {X 103.511,Y 99.686,Z 86.000,A 180.000,B 0.000,C 180.000} C_DIS
LIN {X 103.552,Y 99.578,Z 86.000,A 180.000,B 0.000,C 180.000} C_DIS
LIN {X 103.610,Y 99.399,Z 86.000,A 180.000,B 0.000,C 180.000} C_DIS
LIN {X 103.660,Y 99.221,Z 86.000,A 180.000,B 0.000,C 180.000} C_DIS
LIN {X 103.690,Y 99.103,Z 86.000,A 180.000,B 0.000,C 180.000} C_DIS
LIN {X 103.706,Y 99.042,Z 86.000,A 180.000,B 0.000,C 180.000} C_DIS
LIN {X 103.751,Y 98.863,Z 86.000,A 180.000,B 0.000,C 180.000} C_DIS
LIN {X 103.788,Y 98.684,Z 86.000,A 180.000,B 0.000,C 180.000} C_DIS
LIN {X 103.817,Y 98.505,Z 86.000,A 180.000,B 0.000,C 180.000} C_DIS
LIN {X 103.841,Y 98.327,Z 86.000,A 180.000,B 0.000,C 180.000} C_DIS
LIN {X 103.863,Y 98.148,Z 86.000,A 180.000,B 0.000,C 180.000} C_DIS
LIN {X 103.869,Y 98.105,Z 86.000,A 180.000,B 0.000,C 180.000} C_DIS
LIN {X 103.881,Y 97.969,Z 86.000,A 180.000,B 0.000,C 180.000} C_DIS
LIN {X 103.891,Y 97.790,Z 86.000,A 180.000,B 0.000,C 180.000} C_DIS
LIN {X 103.895,Y 97.612,Z 86.000,A 180.000,B 0.000,C 180.000} C_DIS
LIN {X 103.895,Y 97.433,Z 86.000,A 180.000,B 0.000,C 180.000} C_DIS
LIN {X 103.893,Y 97.254,Z 86.000,A 180.000,B 0.000,C 180.000} C_DIS
LIN {X 103.885,Y 97.075,Z 86.000,A 180.000,B 0.000,C 180.000} C_DIS
LIN {X 103.869,Y 96.897,Z 86.000,A 180.000,B 0.000,C 180.000} C_DIS
LIN {X 103.869,Y 96.895,Z 86.000,A 180.000,B 0.000,C 180.000} C_DIS
LIN {X 103.847,Y 96.718,Z 86.000,A 180.000,B 0.000,C 180.000} C_DIS
LIN {X 103.823,Y 96.539,Z 86.000,A 180.000,B 0.000,C 180.000} C_DIS
LIN {X 103.796,Y 96.360,Z 86.000,A 180.000,B 0.000,C 180.000} C_DIS
LIN {X 103.761,Y 96.181,Z 86.000,A 180.000,B 0.000,C 180.000} C_DIS
LIN {X 103.717,Y 96.003,Z 86.000,A 180.000,B 0.000,C 180.000} C_DIS
LIN {X 103.671,Y 95.824,Z 86.000,A 180.000,B 0.000,C 180.000} C_DIS
LIN {X 103.623,Y 95.645,Z 86.000,A 180.000,B 0.000,C 180.000} C_DIS
LIN {X 103.567,Y 95.466,Z 86.000,A 180.000,B 0.000,C 180.000} C_DIS
LIN {X 103.511,Y 95.314,Z 86.000,A 180.000,B 0.000,C 180.000} C_DIS
LIN {X 103.501,Y 95.288,Z 86.000,A 180.000,B 0.000,C 180.000} C_DIS
LIN {X 103.431,Y 95.109,Z 86.000,A 180.000,B 0.000,C 180.000} C_DIS
LIN {X 103.359,Y 94.930,Z 86.000,A 180.000,B 0.000,C 180.000} C_DIS
LIN {X 103.332,Y 94.870,Z 86.000,A 180.000,B 0.000,C 180.000} C_DIS
LIN {X 103.278,Y 94.751,Z 86.000,A 180.000,B 0.000,C 180.000} C_DIS
LIN {X 103.187,Y 94.573,Z 86.000,A 180.000,B 0.000,C 180.000} C_DIS
LIN {X 103.153,Y 94.510,Z 86.000,A 180.000,B 0.000,C 180.000} C_DIS
LIN {X 103.090,Y 94.394,Z 86.000,A 180.000,B 0.000,C 180.000} C_DIS
LIN {X 102.989,Y 94.215,Z 86.000,A 180.000,B 0.000,C 180.000} C_DIS
LIN {X 102.975,Y 94.190,Z 86.000,A 180.000,B 0.000,C 180.000} C_DIS
LIN {X 102.880,Y 94.036,Z 86.000,A 180.000,B 0.000,C 180.000} C_DIS
LIN {X 102.796,Y 93.911,Z 86.000,A 180.000,B 0.000,C 180.000} C_DIS
LIN {X 102.758,Y 93.857,Z 86.000,A 180.000,B 0.000,C 180.000} C_DIS
LIN {X 102.617,Y 93.664,Z 86.000,A 180.000,B 0.000,C 180.000} C_DIS
LIN {X 102.494,Y 93.500,Z 86.000,A 180.000,B 0.000,C 180.000} C_DIS
LIN {X 102.438,Y 93.431,Z 86.000,A 180.000,B 0.000,C 180.000} C_DIS
LIN {X 102.345,Y 93.321,Z 86.000,A 180.000,B 0.000,C 180.000} C_DIS
LIN {X 102.260,Y 93.228,Z 86.000,A 180.000,B 0.000,C 180.000} C_DIS
LIN {X 102.179,Y 93.142,Z 86.000,A 180.000,B 0.000,C 180.000} C_DIS
LIN {X 102.081,Y 93.038,Z 86.000,A 180.000,B 0.000,C 180.000} C_DIS
LIN {X 102.011,Y 92.964,Z 86.000,A 180.000,B 0.000,C 180.000} C_DIS
LIN {X 101.902,Y 92.857,Z 86.000,A 180.000,B 0.000,C 180.000} C_DIS
LIN {X 101.825,Y 92.785,Z 86.000,A 180.000,B 0.000,C 180.000} C_DIS
LIN {X 101.723,Y 92.696,Z 86.000,A 180.000,B 0.000,C 180.000} C_DIS
LIN {X 101.616,Y 92.606,Z 86.000,A 180.000,B 0.000,C 180.000} C_DIS
LIN {X 101.545,Y 92.547,Z 86.000,A 180.000,B 0.000,C 180.000} C_DIS
LIN {X 101.399,Y 92.427,Z 86.000,A 180.000,B 0.000,C 180.000} C_DIS
LIN {X 101.366,Y 92.402,Z 86.000,A 180.000,B 0.000,C 180.000} C_DIS
LIN {X 101.187,Y 92.271,Z 86.000,A 180.000,B 0.000,C 180.000} C_DIS
LIN {X 101.154,Y 92.249,Z 86.000,A 180.000,B 0.000,C 180.000} C_DIS
LIN {X 101.008,Y 92.153,Z 86.000,A 180.000,B 0.000,C 180.000} C_DIS
LIN {X 100.829,Y 92.039,Z 86.000,A 180.000,B 0.000,C 180.000} C_DIS
LIN {X 100.651,Y 91.931,Z 86.000,A 180.000,B 0.000,C 180.000} C_DIS
LIN {X 100.580,Y 91.891,Z 86.000,A 180.000,B 0.000,C 180.000} C_DIS
LIN {X 100.472,Y 91.835,Z 86.000,A 180.000,B 0.000,C 180.000} C_DIS
LIN {X 100.293,Y 91.747,Z 86.000,A 180.000,B 0.000,C 180.000} C_DIS
LIN {X 100.114,Y 91.663,Z 86.000,A 180.000,B 0.000,C 180.000} C_DIS
LIN {X 99.936,Y 91.583,Z 86.000,A 180.000,B 0.000,C 180.000} C_DIS
LIN {X 99.810,Y 91.533,Z 86.000,A 180.000,B 0.000,C 180.000} C_DIS
LIN {X 99.757,Y 91.513,Z 86.000,A 180.000,B 0.000,C 180.000} C_DIS
LIN {X 99.578,Y 91.452,Z 86.000,A 180.000,B 0.000,C 180.000} C_DIS
LIN {X 99.399,Y 91.394,Z 86.000,A 180.000,B 0.000,C 180.000} C_DIS
LIN {X 99.277,Y 91.355,Z 86.000,A 180.000,B 0.000,C 180.000} C_DIS
LIN {X 99.221,Y 91.337,Z 86.000,A 180.000,B 0.000,C 180.000} C_DIS
LIN {X 99.042,Y 91.290,Z 86.000,A 180.000,B 0.000,C 180.000} C_DIS
LIN {X 98.863,Y 91.251,Z 86.000,A 180.000,B 0.000,C 180.000} C_DIS
LIN {X 98.684,Y 91.216,Z 86.000,A 180.000,B 0.000,C 180.000} C_DIS
LIN {X 98.505,Y 91.182,Z 86.000,A 180.000,B 0.000,C 180.000} C_DIS
LIN {X 98.468,Y 91.176,Z 86.000,A 180.000,B 0.000,C 180.000} C_DIS
LIN {X 98.327,Y 91.155,Z 86.000,A 180.000,B 0.000,C 180.000} C_DIS
LIN {X 98.148,Y 91.136,Z 86.000,A 180.000,B 0.000,C 180.000} C_DIS
LIN {X 97.969,Y 91.122,Z 86.000,A 180.000,B 0.000,C 180.000} C_DIS
LIN {X 97.790,Y 91.111,Z 86.000,A 180.000,B 0.000,C 180.000} C_DIS
LIN {X 97.612,Y 91.103,Z 86.000,A 180.000,B 0.000,C 180.000} C_DIS
LIN {X 97.433,Y 91.102,Z 86.000,A 180.000,B 0.000,C 180.000} C_DIS
LIN {X 97.254,Y 91.108,Z 86.000,A 180.000,B 0.000,C 180.000} C_DIS
LIN {X 97.075,Y 91.119,Z 86.000,A 180.000,B 0.000,C 180.000} C_DIS
LIN {X 96.897,Y 91.132,Z 86.000,A 180.000,B 0.000,C 180.000} C_DIS
LIN {X 96.718,Y 91.149,Z 86.000,A 180.000,B 0.000,C 180.000} C_DIS
LIN {X 96.539,Y 91.175,Z 86.000,A 180.000,B 0.000,C 180.000} C_DIS
LIN {X 96.532,Y 91.176,Z 86.000,A 180.000,B 0.000,C 180.000} C_DIS
LIN {X 96.360,Y 91.208,Z 86.000,A 180.000,B 0.000,C 180.000} C_DIS
LIN {X 96.181,Y 91.242,Z 86.000,A 180.000,B 0.000,C 180.000} C_DIS
LIN {X 96.003,Y 91.279,Z 86.000,A 180.000,B 0.000,C 180.000} C_DIS
LIN {X 95.824,Y 91.325,Z 86.000,A 180.000,B 0.000,C 180.000} C_DIS
LIN {X 95.723,Y 91.355,Z 86.000,A 180.000,B 0.000,C 180.000} C_DIS
LIN {X 95.645,Y 91.380,Z 86.000,A 180.000,B 0.000,C 180.000} C_DIS
LIN {X 95.466,Y 91.437,Z 86.000,A 180.000,B 0.000,C 180.000} C_DIS
LIN {X 95.288,Y 91.497,Z 86.000,A 180.000,B 0.000,C 180.000} C_DIS
LIN {X 95.190,Y 91.533,Z 86.000,A 180.000,B 0.000,C 180.000} C_DIS
LIN {X 95.109,Y 91.565,Z 86.000,A 180.000,B 0.000,C 180.000} C_DIS
LIN {X 94.930,Y 91.643,Z 86.000,A 180.000,B 0.000,C 180.000} C_DIS
LIN {X 94.781,Y 91.712,Z 86.000,A 180.000,B 0.000,C 180.000} C_DIS
LIN {X 94.751,Y 91.726,Z 86.000,A 180.000,B 0.000,C 180.000} C_DIS
LIN {X 94.573,Y 91.812,Z 86.000,A 180.000,B 0.000,C 180.000} C_DIS
LIN {X 94.420,Y 91.891,Z 86.000,A 180.000,B 0.000,C 180.000} C_DIS
LIN {X 94.394,Y 91.906,Z 86.000,A 180.000,B 0.000,C 180.000} C_DIS
LIN {X 94.215,Y 92.011,Z 86.000,A 180.000,B 0.000,C 180.000} C_DIS
LIN {X 94.123,Y 92.070,Z 86.000,A 180.000,B 0.000,C 180.000} C_DIS
LIN {X 94.036,Y 92.125,Z 86.000,A 180.000,B 0.000,C 180.000} C_DIS
LIN {X 93.857,Y 92.241,Z 86.000,A 180.000,B 0.000,C 180.000} C_DIS
LIN {X 93.846,Y 92.249,Z 86.000,A 180.000,B 0.000,C 180.000} C_DIS
LIN {X 93.679,Y 92.369,Z 86.000,A 180.000,B 0.000,C 180.000} C_DIS
LIN {X 93.601,Y 92.427,Z 86.000,A 180.000,B 0.000,C 180.000} C_DIS
LIN {X 93.500,Y 92.510,Z 86.000,A 180.000,B 0.000,C 180.000} C_DIS
LIN {X 93.384,Y 92.606,Z 86.000,A 180.000,B 0.000,C 180.000} C_DIS
LIN {X 93.321,Y 92.658,Z 86.000,A 180.000,B 0.000,C 180.000} C_DIS
LIN {X 93.175,Y 92.785,Z 86.000,A 180.000,B 0.000,C 180.000} C_DIS
LIN {X 93.142,Y 92.815,Z 86.000,A 180.000,B 0.000,C 180.000} C_DIS
LIN {X 92.989,Y 92.964,Z 86.000,A 180.000,B 0.000,C 180.000} C_DIS
LIN {X 92.964,Y 92.991,Z 86.000,A 180.000,B 0.000,C 180.000} C_DIS
LIN {X 92.821,Y 93.142,Z 86.000,A 180.000,B 0.000,C 180.000} C_DIS
LIN {X 92.785,Y 93.180,Z 86.000,A 180.000,B 0.000,C 180.000} C_DIS
LIN {X 92.655,Y 93.321,Z 86.000,A 180.000,B 0.000,C 180.000} C_DIS
LIN {X 92.606,Y 93.379,Z 86.000,A 180.000,B 0.000,C 180.000} C_DIS
LIN {X 92.506,Y 93.500,Z 86.000,A 180.000,B 0.000,C 180.000} C_DIS
LIN {X 92.427,Y 93.604,Z 86.000,A 180.000,B 0.000,C 180.000} C_DIS
LIN {X 92.372,Y 93.679,Z 86.000,A 180.000,B 0.000,C 180.000} C_DIS
LIN {X 92.242,Y 93.857,Z 86.000,A 180.000,B 0.000,C 180.000} C_DIS
LIN {X 92.120,Y 94.036,Z 86.000,A 180.000,B 0.000,C 180.000} C_DIS
LIN {X 92.070,Y 94.115,Z 86.000,A 180.000,B 0.000,C 180.000} C_DIS
LIN {X 92.011,Y 94.215,Z 86.000,A 180.000,B 0.000,C 180.000} C_DIS
LIN {X 91.910,Y 94.394,Z 86.000,A 180.000,B 0.000,C 180.000} C_DIS
LIN {X 91.891,Y 94.429,Z 86.000,A 180.000,B 0.000,C 180.000} C_DIS
LIN {X 91.813,Y 94.573,Z 86.000,A 180.000,B 0.000,C 180.000} C_DIS
LIN {X 91.722,Y 94.751,Z 86.000,A 180.000,B 0.000,C 180.000} C_DIS
LIN {X 91.712,Y 94.771,Z 86.000,A 180.000,B 0.000,C 180.000} C_DIS
LIN {X 91.641,Y 94.930,Z 86.000,A 180.000,B 0.000,C 180.000} C_DIS
LIN {X 91.569,Y 95.109,Z 86.000,A 180.000,B 0.000,C 180.000} C_DIS
LIN {X 91.533,Y 95.199,Z 86.000,A 180.000,B 0.000,C 180.000} C_DIS
LIN {X 91.499,Y 95.288,Z 86.000,A 180.000,B 0.000,C 180.000} C_DIS
LIN {X 91.433,Y 95.466,Z 86.000,A 180.000,B 0.000,C 180.000} C_DIS
LIN {X 91.377,Y 95.645,Z 86.000,A 180.000,B 0.000,C 180.000} C_DIS
LIN {X 91.355,Y 95.724,Z 86.000,A 180.000,B 0.000,C 180.000} C_DIS
LIN {X 91.329,Y 95.824,Z 86.000,A 180.000,B 0.000,C 180.000} C_DIS
LIN {X 91.283,Y 96.003,Z 86.000,A 180.000,B 0.000,C 180.000} C_DIS
LIN {X 91.239,Y 96.181,Z 86.000,A 180.000,B 0.000,C 180.000} C_DIS
LIN {X 91.204,Y 96.360,Z 86.000,A 180.000,B 0.000,C 180.000} C_DIS
LIN {X 91.177,Y 96.539,Z 86.000,A 180.000,B 0.000,C 180.000} C_DIS
LIN {X 91.176,Y 96.543,Z 86.000,A 180.000,B 0.000,C 180.000} C_DIS
LIN {X 91.168,Y 96.604,Z 86.000,A 180.000,B 0.000,C 180.000} C_DIS
; Link Move Starts
LIN {X 91.130,Y 96.911,Z 86.000,A 180.000,B 0.000,C 180.000} C_DIS
LIN {X 91.109,Y 97.190,Z 85.999,A 180.000,B 0.000,C 180.000} C_DIS
LIN {X 91.104,Y 97.487,Z 85.998,A 180.000,B 0.000,C 180.000} C_DIS
LIN {X 91.107,Y 97.779,Z 85.997,A 180.000,B 0.000,C 180.000} C_DIS
LIN {X 91.126,Y 98.076,Z 85.995,A 180.000,B 0.000,C 180.000} C_DIS
LIN {X 91.161,Y 98.370,Z 85.992,A 180.000,B 0.000,C 180.000} C_DIS
LIN {X 91.201,Y 98.653,Z 85.990,A 180.000,B 0.000,C 180.000} C_DIS
LIN {X 91.260,Y 98.934,Z 85.987,A 180.000,B 0.000,C 180.000} C_DIS
LIN {X 91.337,Y 99.239,Z 85.983,A 180.000,B 0.000,C 180.000} C_DIS
LIN {X 91.417,Y 99.515,Z 85.979,A 180.000,B 0.000,C 180.000} C_DIS
LIN {X 91.514,Y 99.784,Z 85.975,A 180.000,B 0.000,C 180.000} C_DIS
LIN {X 91.625,Y 100.068,Z 85.971,A 180.000,B 0.000,C 180.000} C_DIS
LIN {X 91.742,Y 100.326,Z 85.966,A 180.000,B 0.000,C 180.000} C_DIS
LIN {X 91.810,Y 100.460,Z 85.963,A 180.000,B 0.000,C 180.000} C_DIS
LIN {X 91.882,Y 100.593,Z 85.961,A 180.000,B 0.000,C 180.000} C_DIS
LIN {X 91.952,Y 100.723,Z 85.958,A 180.000,B 0.000,C 180.000} C_DIS
LIN {X 92.025,Y 100.851,Z 85.955,A 180.000,B 0.000,C 180.000} C_DIS
LIN {X 92.102,Y 100.977,Z 85.952,A 180.000,B 0.000,C 180.000} C_DIS
LIN {X 92.183,Y 101.100,Z 85.949,A 180.000,B 0.000,C 180.000} C_DIS
LIN {X 92.268,Y 101.220,Z 85.946,A 180.000,B 0.000,C 180.000} C_DIS
LIN {X 92.353,Y 101.340,Z 85.943,A 180.000,B 0.000,C 180.000} C_DIS
LIN {X 92.441,Y 101.461,Z 85.940,A 180.000,B 0.000,C 180.000} C_DIS
LIN {X 92.531,Y 101.579,Z 85.936,A 180.000,B 0.000,C 180.000} C_DIS
LIN {X 92.621,Y 101.687,Z 85.933,A 180.000,B 0.000,C 180.000} C_DIS
LIN {X 92.714,Y 101.792,Z 85.930,A 180.000,B 0.000,C 180.000} C_DIS
LIN {X 92.817,Y 101.904,Z 85.926,A 180.000,B 0.000,C 180.000} C_DIS
LIN {X 92.921,Y 102.017,Z 85.923,A 180.000,B 0.000,C 180.000} C_DIS
LIN {X 93.022,Y 102.123,Z 85.919,A 180.000,B 0.000,C 180.000} C_DIS
LIN {X 93.127,Y 102.225,Z 85.915,A 180.000,B 0.000,C 180.000} C_DIS
LIN {X 93.236,Y 102.324,Z 85.911,A 180.000,B 0.000,C 180.000} C_DIS
LIN {X 93.348,Y 102.420,Z 85.907,A 180.000,B 0.000,C 180.000} C_DIS
LIN {X 93.464,Y 102.518,Z 85.903,A 180.000,B 0.000,C 180.000} C_DIS
LIN {X 93.581,Y 102.616,Z 85.899,A 180.000,B 0.000,C 180.000} C_DIS
LIN {X 93.693,Y 102.704,Z 85.895,A 180.000,B 0.000,C 180.000} C_DIS
LIN {X 93.809,Y 102.788,Z 85.891,A 180.000,B 0.000,C 180.000} C_DIS
LIN {X 93.933,Y 102.873,Z 85.887,A 180.000,B 0.000,C 180.000} C_DIS
LIN {X 94.060,Y 102.955,Z 85.883,A 180.000,B 0.000,C 180.000} C_DIS
LIN {X 94.185,Y 103.037,Z 85.878,A 180.000,B 0.000,C 180.000} C_DIS
LIN {X 94.312,Y 103.115,Z 85.874,A 180.000,B 0.000,C 180.000} C_DIS
LIN {X 94.439,Y 103.188,Z 85.869,A 180.000,B 0.000,C 180.000} C_DIS
LIN {X 94.569,Y 103.257,Z 85.865,A 180.000,B 0.000,C 180.000} C_DIS
LIN {X 94.703,Y 103.323,Z 85.860,A 180.000,B 0.000,C 180.000} C_DIS
LIN {X 94.837,Y 103.389,Z 85.855,A 180.000,B 0.000,C 180.000} C_DIS
LIN {X 94.967,Y 103.450,Z 85.851,A 180.000,B 0.000,C 180.000} C_DIS
LIN {X 95.099,Y 103.508,Z 85.846,A 180.000,B 0.000,C 180.000} C_DIS
LIN {X 95.238,Y 103.564,Z 85.841,A 180.000,B 0.000,C 180.000} C_DIS
LIN {X 95.379,Y 103.614,Z 85.836,A 180.000,B 0.000,C 180.000} C_DIS
LIN {X 95.451,Y 103.639,Z 85.834,A 180.000,B 0.000,C 180.000} C_DIS
LIN {X 95.524,Y 103.664,Z 85.831,A 180.000,B 0.000,C 180.000} C_DIS
LIN {X 95.597,Y 103.689,Z 85.829,A 180.000,B 0.000,C 180.000} C_DIS
LIN {X 95.669,Y 103.713,Z 85.826,A 180.000,B 0.000,C 180.000} C_DIS
LIN {X 95.805,Y 103.756,Z 85.821,A 180.000,B 0.000,C 180.000} C_DIS
LIN {X 95.942,Y 103.794,Z 85.816,A 180.000,B 0.000,C 180.000} C_DIS
LIN {X 96.015,Y 103.813,Z 85.814,A 180.000,B 0.000,C 180.000} C_DIS
LIN {X 96.089,Y 103.829,Z 85.811,A 180.000,B 0.000,C 180.000} C_DIS
LIN {X 96.162,Y 103.845,Z 85.808,A 180.000,B 0.000,C 180.000} C_DIS
LIN {X 96.236,Y 103.861,Z 85.806,A 180.000,B 0.000,C 180.000} C_DIS
LIN {X 96.385,Y 103.892,Z 85.800,A 180.000,B 0.000,C 180.000} C_DIS
LIN {X 96.460,Y 103.907,Z 85.798,A 180.000,B 0.000,C 180.000} C_DIS
LIN {X 96.535,Y 103.922,Z 85.795,A 180.000,B 0.000,C 180.000} C_DIS
LIN {X 96.677,Y 103.944,Z 85.790,A 180.000,B 0.000,C 180.000} C_DIS
LIN {X 96.748,Y 103.954,Z 85.787,A 180.000,B 0.000,C 180.000} C_DIS
LIN {X 96.820,Y 103.962,Z 85.785,A 180.000,B 0.000,C 180.000} C_DIS
LIN {X 96.895,Y 103.970,Z 85.782,A 180.000,B 0.000,C 180.000} C_DIS
LIN {X 96.971,Y 103.977,Z 85.780,A 180.000,B 0.000,C 180.000} C_DIS
LIN {X 97.199,Y 103.995,Z 85.772,A 180.000,B 0.000,C 180.000} C_DIS
LIN {X 97.275,Y 104.001,Z 85.769,A 180.000,B 0.000,C 180.000} C_DIS
LIN {X 97.351,Y 104.005,Z 85.766,A 180.000,B 0.000,C 180.000} C_DIS
LIN {X 97.427,Y 104.008,Z 85.764,A 180.000,B 0.000,C 180.000} C_DIS
LIN {X 97.500,Y 104.010,Z 85.761,A 180.000,B 0.000,C 180.000} C_DIS
LIN {X 97.573,Y 104.010,Z 85.759,A 180.000,B 0.000,C 180.000} C_DIS
LIN {X 97.645,Y 104.010,Z 85.756,A 180.000,B 0.000,C 180.000} C_DIS
LIN {X 97.718,Y 104.008,Z 85.754,A 180.000,B 0.000,C 180.000} C_DIS
LIN {X 97.794,Y 104.005,Z 85.751,A 180.000,B 0.000,C 180.000} C_DIS
LIN {X 97.945,Y 103.998,Z 85.746,A 180.000,B 0.000,C 180.000} C_DIS
LIN {X 98.021,Y 103.995,Z 85.743,A 180.000,B 0.000,C 180.000} C_DIS
